  Call Extruder(12670.239)
  MoveL 1268 to (9.47, 41.51, 60) mm, rotated rx 180 ry 0 rz 180 deg; joints [36.675, 60.104, 7.721, -141.195, 72.379, -193.682]
  Call Extruder(12685.135)
  MoveL 1269 to (0, 42.57, 60) mm, rotated rx 180 ry 0 rz 180 deg; joints [37.594, 59.268, 9.663, -140.474, 73.45, -193.226]
  Call Extruder(12700.031)
  MoveL 1270 to (-9.47, 41.5, 60) mm, rotated rx -180 ry 0 rz 180 deg; joints [38.304, 58.316, 11.901, -139.989, 74.597, -192.569]
  Call Extruder(12714.927)
  MoveL 1271 to (-18.47, 38.36, 60) mm, rotated rx 180 ry 0 rz 180 deg; joints [38.762, 57.3, 14.324, -139.766, 75.77, -191.749]
  Call Extruder(12729.823)
  MoveL 1272 to (-26.54, 33.28, 60) mm, rotated rx -180 ry 0 rz 180 deg; joints [38.928, 56.273, 16.816, -139.828, 76.922, -190.815]
  Call Extruder(12744.719)
  MoveL 1273 to (-33.29, 26.54, 60) mm, rotated rx 180 ry 0 rz 180 deg; joints [38.772, 55.287, 19.256, -140.194, 78.008, -189.824]
  Call Extruder(12759.614)
  MoveL 1274 to (-38.36, 18.47, 60) mm, rotated rx 180 ry 0 rz 180 deg; joints [38.277, 54.389, 21.525, -140.869, 78.986, -188.835]
  Call Extruder(12774.510)
  MoveL 1275 to (-41.51, 9.47, 60) mm, rotated rx 180 ry 0 rz 180 deg; joints [37.447, 53.619, 23.509, -141.847, 79.813, -187.91]
  Call Extruder(12789.406)
  MoveL 1276 to (-42.57, 0, 60) mm, rotated rx 180 ry 0 rz 180 deg; joints [36.31, 53.012, 25.105, -143.096, 80.448, -187.103]
  Call Extruder(12796.960)
  MoveL 1277 to (-42.03, -4.8, 60) mm, rotated rx 180 ry 0 rz 180 deg; joints [35.612, 52.795, 25.681, -143.834, 80.653, -186.771]
  Set speed (130.0 mm/s)
  MoveL 1278 to (-54.1, -7.67, 60) mm, rotated rx 180 ry 0 rz -180 deg; joints [36.421, 51.788, 28.414, -143.176, 82.129, -185.854]
  Call Extruder(12801.033)
  Set speed (30.0 mm/s)
  MoveL 1279 to (-53.59, -12.23, 60) mm, rotated rx 180 ry 0 rz 180 deg; joints [35.732, 51.595, 28.949, -143.896, 82.336, -185.556]
  Call Extruder(12811.963)
  MoveL 1280 to (-49.53, -23.85, 60) mm, rotated rx 180 ry 0 rz 180 deg; joints [33.663, 51.321, 29.715, -146.012, 82.549, -184.997]
  Call Extruder(12822.893)
  MoveL 1281 to (-42.98, -34.27, 60) mm, rotated rx -180 ry 0 rz -180 deg; joints [31.506, 51.313, 29.737, -148.181, 82.378, -184.705]
  Call Extruder(12833.823)
  MoveL 1282 to (-34.27, -42.98, 60) mm, rotated rx -180 ry 0 rz -180 deg; joints [29.427, 51.572, 29.014, -150.24, 81.809, -184.657]
  Call Extruder(12844.754)
  MoveL 1283 to (-23.85, -49.53, 60) mm, rotated rx 180 ry 0 rz 180 deg; joints [27.581, 52.088, 27.588, -152.034, 80.86, -184.821]
  Call Extruder(12855.684)
  MoveL 1284 to (-12.23, -53.59, 60) mm, rotated rx 180 ry 0 rz 180 deg; joints [26.087, 52.846, 25.544, -153.443, 79.587, -185.162]
  Call Extruder(12866.614)
  MoveL 1285 to (0, -54.97, 60) mm, rotated rx 180 ry 0 rz 180 deg; joints [25.019, 53.817, 22.995, -154.389, 78.069, -185.66]
  Call Extruder(12870.401)
  MoveL 1286 to (4.24, -54.49, 60) mm, rotated rx 180 ry 0 rz 180 deg; joints [24.802, 54.206, 21.993, -154.553, 77.494, -185.883]
  Call Extruder(12877.544)
  MoveL 1287 to (12.23, -53.59, 60) mm, rotated rx 180 ry 0 rz 180 deg; joints [24.406, 54.961, 20.076, -154.842, 76.4, -186.302]
  Call Extruder(12888.474)
  MoveL 1288 to (23.85, -49.53, 60) mm, rotated rx -180 ry 0 rz 180 deg; joints [24.239, 56.226, 16.932, -154.807, 74.681, -187.084]
  Call Extruder(12899.405)
  MoveL 1289 to (34.27, -42.98, 60) mm, rotated rx -180 ry 0 rz 180 deg; joints [24.487, 57.553, 13.715, -154.316, 73.007, -188.001]
  Call Extruder(12910.335)
  MoveL 1290 to (42.98, -34.27, 60) mm, rotated rx 180 ry 0 rz 180 deg; joints [25.101, 58.878, 10.576, -153.422, 71.469, -189.035]
  Call Extruder(12921.265)
  MoveL 1291 to (49.52, -23.85, 60) mm, rotated rx 180 ry 0 rz 180 deg; joints [26.025, 60.129, 7.663, -152.193, 70.145, -190.155]
  Call Extruder(12932.195)
  MoveL 1292 to (53.59, -12.23, 60) mm, rotated rx -180 ry 0 rz 180 deg; joints [27.2, 61.238, 5.12, -150.706, 69.104, -191.316]
  Call Extruder(12943.125)
  MoveL 1293 to (54.97, 0, 60) mm, rotated rx 180 ry 0 rz 180 deg; joints [28.57, 62.141, 3.074, -149.045, 68.397, -192.452]
  Call Extruder(12954.056)
  MoveL 1294 to (53.59, 12.23, 60) mm, rotated rx 180 ry 0 rz 180 deg; joints [30.077, 62.781, 1.635, -147.296, 68.057, -193.492]
  Call Extruder(12964.986)
  MoveL 1295 to (49.52, 23.85, 60) mm, rotated rx 180 ry 0 rz 180 deg; joints [31.665, 63.117, 0.883, -145.541, 68.093, -194.361]
  Call Extruder(12975.916)
  MoveL 1296 to (42.98, 34.27, 60) mm, rotated rx 180 ry 0 rz 180 deg; joints [33.282, 63.127, 0.862, -143.855, 68.493, -194.991]
  Call Extruder(12986.846)
  MoveL 1297 to (34.27, 42.98, 60) mm, rotated rx 180 ry 0 rz -180 deg; joints [34.874, 62.81, 1.571, -142.299, 69.223, -195.333]
  Call Extruder(12997.776)
  MoveL 1298 to (23.85, 49.53, 60) mm, rotated rx -180 ry 0 rz 180 deg; joints [36.387, 62.186, 2.972, -140.922, 70.232, -195.357]
  Call Extruder(13008.707)
  MoveL 1299 to (12.23, 53.59, 60) mm, rotated rx 180 ry 0 rz 180 deg; joints [37.766, 61.298, 4.984, -139.762, 71.46, -195.06]
  Call Extruder(13019.637)
  MoveL 1300 to (0, 54.97, 60) mm, rotated rx 180 ry 0 rz 180 deg; joints [38.954, 60.199, 7.502, -138.852, 72.838, -194.458]
  Call Extruder(13030.567)
  MoveL 1301 to (-12.23, 53.59, 60) mm, rotated rx -180 ry 0 rz -180 deg; joints [39.895, 58.954, 10.397, -138.223, 74.302, -193.588]
  Call Extruder(13041.497)
  MoveL 1302 to (-23.85, 49.53, 60) mm, rotated rx 180 ry 0 rz 180 deg; joints [40.528, 57.632, 13.527, -137.907, 75.791, -192.502]
  Call Extruder(13052.427)
  MoveL 1303 to (-34.27, 42.98, 60) mm, rotated rx 180 ry 0 rz 180 deg; joints [40.799, 56.303, 16.743, -137.938, 77.247, -191.265]
  Call Extruder(13063.358)
  MoveL 1304 to (-42.98, 34.27, 60) mm, rotated rx 180 ry 0 rz 180 deg; joints [40.659, 55.032, 19.896, -138.348, 78.623, -189.952]
  Call Extruder(13074.288)
  MoveL 1305 to (-49.53, 23.85, 60) mm, rotated rx -180 ry 0 rz -180 deg; joints [40.072, 53.88, 22.832, -139.16, 79.87, -188.645]
  Call Extruder(13085.218)
  MoveL 1306 to (-53.59, 12.23, 60) mm, rotated rx 180 ry 0 rz 180 deg; joints [39.031, 52.898, 25.406, -140.38, 80.94, -187.427]
  Call Extruder(13096.148)
  MoveL 1307 to (-54.97, 0, 60) mm, rotated rx 180 ry 0 rz 180 deg; joints [37.56, 52.127, 27.484, -141.981, 81.781, -186.377]
  Call Extruder(13101.674)
  MoveL 1308 to (-54.27, -6.18, 60) mm, rotated rx 180 ry 0 rz -180 deg; joints [36.644, 51.852, 28.237, -142.942, 82.062, -185.954]
  Set speed (130.0 mm/s)
  MoveL 1309 to (-49.9, -9.51, 60) mm, rotated rx -180 ry 0 rz -180 deg; joints [35.741, 51.987, 27.866, -143.829, 81.779, -185.968]
  MoveL 1310 to (2.97, -12.99, 60) mm, rotated rx 180 ry 0 rz 180 deg; joints [30.614, 56.045, 17.377, -148.309, 75.785, -188.621]
  Call Extruder(13106.337)
  Set speed (80.0 mm/s)
  MoveL 1311 to (5.78, -12.01, 60) mm, rotated rx -180 ry 0 rz -180 deg; joints [30.526, 56.355, 16.616, -148.338, 75.388, -188.843]
  Call Extruder(13111.001)
  MoveL 1312 to (8.31, -10.42, 60) mm, rotated rx 180 ry 0 rz -180 deg; joints [30.538, 56.675, 15.835, -148.261, 74.998, -189.096]
  Call Extruder(13115.665)
  MoveL 1313 to (10.42, -8.31, 60) mm, rotated rx 180 ry 0 rz 180 deg; joints [30.649, 56.989, 15.074, -148.084, 74.636, -189.37]
  Call Extruder(13120.329)
  MoveL 1314 to (12.01, -5.78, 60) mm, rotated rx 180 ry 0 rz 180 deg; joints [30.85, 57.281, 14.369, -147.817, 74.319, -189.653]
  Call Extruder(13124.992)
  MoveL 1315 to (12.99, -2.97, 60) mm, rotated rx 180 ry 0 rz -180 deg; joints [31.131, 57.536, 13.756, -147.476, 74.065, -189.93]
  Call Extruder(13129.656)
  MoveL 1316 to (13.33, 0, 60) mm, rotated rx 180 ry 0 rz -180 deg; joints [31.476, 57.741, 13.266, -147.078, 73.885, -190.188]
  Call Extruder(13134.320)
  MoveL 1317 to (13, 2.97, 60) mm, rotated rx 180 ry 0 rz -180 deg; joints [31.869, 57.885, 12.924, -146.644, 73.789, -190.413]
  Call Extruder(13138.984)
  MoveL 1318 to (12.01, 5.78, 60) mm, rotated rx 180 ry 0 rz -180 deg; joints [32.292, 57.96, 12.745, -146.194, 73.78, -190.594]
  Call Extruder(13143.648)
  MoveL 1319 to (10.42, 8.31, 60) mm, rotated rx 180 ry 0 rz 180 deg; joints [32.725, 57.962, 12.74, -145.75, 73.857, -190.719]
  Call Extruder(13148.312)
  MoveL 1320 to (8.31, 10.42, 60) mm, rotated rx 180 ry 0 rz -180 deg; joints [33.149, 57.891, 12.908, -145.333, 74.017, -190.782]
  Call Extruder(13152.975)
  MoveL 1321 to (5.78, 12.01, 60) mm, rotated rx -180 ry 0 rz -180 deg; joints [33.544, 57.751, 13.242, -144.961, 74.25, -190.777]
  Call Extruder(13157.639)
  MoveL 1322 to (2.97, 13, 60) mm, rotated rx -180 ry 0 rz 180 deg; joints [33.893, 57.55, 13.724, -144.65, 74.544, -190.705]
  Call Extruder(13162.303)
  MoveL 1323 to (0, 13.33, 60) mm, rotated rx 180 ry 0 rz 180 deg; joints [34.177, 57.297, 14.33, -144.416, 74.885, -190.568]
  Call Extruder(13166.967)
  MoveL 1324 to (-2.97, 13, 60) mm, rotated rx 180 ry 0 rz 180 deg; joints [34.384, 57.007, 15.03, -144.27, 75.255, -190.375]
  Call Extruder(13171.630)
  MoveL 1325 to (-5.78, 12.01, 60) mm, rotated rx 180 ry 0 rz -180 deg; joints [34.5, 56.694, 15.79, -144.22, 75.638, -190.136]
  Call Extruder(13176.294)
  MoveL 1326 to (-8.31, 10.42, 60) mm, rotated rx 180 ry 0 rz 180 deg; joints [34.518, 56.374, 16.571, -144.269, 76.015, -189.863]
  Call Extruder(13180.958)
  MoveL 1327 to (-10.42, 8.31, 60) mm, rotated rx 180 ry 0 rz -180 deg; joints [34.436, 56.063, 17.333, -144.417, 76.368, -189.571]
  Call Extruder(13185.622)
  MoveL 1328 to (-12.01, 5.78, 60) mm, rotated rx 180 ry 0 rz 180 deg; joints [34.254, 55.776, 18.04, -144.66, 76.681, -189.278]
  Call Extruder(13190.285)
  MoveL 1329 to (-13, 2.97, 60) mm, rotated rx 180 ry 0 rz 180 deg; joints [33.981, 55.528, 18.655, -144.986, 76.938, -188.997]
  Call Extruder(13194.949)
  MoveL 1330 to (-13.33, 0, 60) mm, rotated rx -180 ry 0 rz -180 deg; joints [33.63, 55.331, 19.148, -145.382, 77.126, -188.744]
  Call Extruder(13199.613)
  MoveL 1331 to (-13, -2.97, 60) mm, rotated rx 180 ry 0 rz -180 deg; joints [33.218, 55.193, 19.493, -145.826, 77.234, -188.532]
  Call Extruder(13204.277)
  MoveL 1332 to (-12.01, -5.78, 60) mm, rotated rx 180 ry 0 rz -180 deg; joints [32.767, 55.121, 19.672, -146.297, 77.258, -188.369]
  Call Extruder(13208.941)
  MoveL 1333 to (-10.42, -8.31, 60) mm, rotated rx 180 ry 0 rz 180 deg; joints [32.302, 55.119, 19.678, -146.769, 77.193, -188.263]
  Call Extruder(13213.605)
  MoveL 1334 to (-8.31, -10.42, 60) mm, rotated rx 180 ry 0 rz -180 deg; joints [31.85, 55.187, 19.508, -147.215, 77.043, -188.218]
  Call Extruder(13218.268)
  MoveL 1335 to (-5.78, -12.01, 60) mm, rotated rx 180 ry 0 rz 180 deg; joints [31.435, 55.321, 19.172, -147.612, 76.814, -188.234]
  Call Extruder(13222.932)
  MoveL 1336 to (-2.97, -12.99, 60) mm, rotated rx 180 ry 0 rz -180 deg; joints [31.079, 55.515, 18.688, -147.937, 76.517, -188.309]
  Call Extruder(13227.596)
  MoveL 1337 to (0, -13.33, 60) mm, rotated rx -180 ry 0 rz 180 deg; joints [30.801, 55.76, 18.079, -148.173, 76.168, -188.44]
  Call Extruder(13232.260)
  MoveL 1338 to (2.97, -12.99, 60) mm, rotated rx 180 ry 0 rz 180 deg; joints [30.614, 56.045, 17.377, -148.309, 75.785, -188.621]
  Set speed (130.0 mm/s)
  MoveL 1339 to (2.97, -13, 65) mm, rotated rx -180 ry 0 rz 180 deg; joints [30.614, 55.122, 17.776, -148.238, 75.34, -188.905]
  MoveL 1340 to (-26.25, -4.54, 65) mm, rotated rx 180 ry 0 rz 180 deg; joints [34.172, 53.056, 22.883, -145.013, 78.404, -188.008]
  Call Extruder(13234.492)
  Set speed (60.0 mm/s)
  MoveL 1341 to (-26.09, -5.96, 65) mm, rotated rx 180 ry 0 rz -180 deg; joints [33.969, 52.991, 23.047, -145.23, 78.457, -187.909]
  Call Extruder(13243.857)
  MoveL 1342 to (-24.12, -11.61, 65) mm, rotated rx 180 ry 0 rz 180 deg; joints [33.033, 52.848, 23.411, -146.202, 78.513, -187.593]
  Call Extruder(13253.222)
  MoveL 1343 to (-20.93, -16.69, 65) mm, rotated rx 180 ry 0 rz -180 deg; joints [32.066, 52.844, 23.422, -147.182, 78.393, -187.393]
  Call Extruder(13262.587)
  MoveL 1344 to (-16.69, -20.93, 65) mm, rotated rx 180 ry 0 rz -180 deg; joints [31.126, 52.979, 23.078, -148.11, 78.096, -187.313]
  Call Extruder(13271.952)
  MoveL 1345 to (-11.61, -24.11, 65) mm, rotated rx 180 ry 0 rz 180 deg; joints [30.272, 53.248, 22.399, -148.931, 77.638, -187.35]
  Call Extruder(13281.317)
  MoveL 1346 to (-5.96, -26.09, 65) mm, rotated rx 180 ry 0 rz -180 deg; joints [29.552, 53.639, 21.419, -149.595, 77.039, -187.498]
  Call Extruder(13290.682)
  MoveL 1347 to (0, -26.77, 65) mm, rotated rx -180 ry 0 rz -180 deg; joints [29.003, 54.134, 20.191, -150.067, 76.332, -187.748]
  Call Extruder(13293.068)
  MoveL 1348 to (1.52, -26.59, 65) mm, rotated rx 180 ry 0 rz 180 deg; joints [28.912, 54.28, 19.832, -150.134, 76.135, -187.835]
  Call Extruder(13300.047)
  MoveL 1349 to (5.96, -26.09, 65) mm, rotated rx 180 ry 0 rz -180 deg; joints [28.65, 54.711, 18.776, -150.323, 75.556, -188.09]
  Call Extruder(13309.412)
  MoveL 1350 to (11.61, -24.12, 65) mm, rotated rx 180 ry 0 rz 180 deg; joints [28.503, 55.341, 17.247, -150.356, 74.753, -188.512]
  Call Extruder(13318.777)
  MoveL 1351 to (16.69, -20.93, 65) mm, rotated rx 180 ry 0 rz 180 deg; joints [28.559, 55.994, 15.679, -150.171, 73.968, -188.998]
  Call Extruder(13328.142)
  MoveL 1352 to (20.93, -16.69, 65) mm, rotated rx 180 ry 0 rz 180 deg; joints [28.808, 56.638, 14.15, -149.785, 73.241, -189.532]
  Call Extruder(13337.507)
  MoveL 1353 to (24.12, -11.61, 65) mm, rotated rx -180 ry 0 rz 180 deg; joints [29.229, 57.24, 12.735, -149.224, 72.612, -190.091]
  Call Extruder(13346.872)
  MoveL 1354 to (26.09, -5.96, 65) mm, rotated rx -180 ry 0 rz -180 deg; joints [29.796, 57.767, 11.505, -148.523, 72.113, -190.65]
  Call Extruder(13356.237)
  MoveL 1355 to (26.77, 0, 65) mm, rotated rx -180 ry 0 rz -180 deg; joints [30.482, 58.192, 10.52, -147.719, 71.767, -191.181]
  Call Extruder(13365.602)
  MoveL 1356 to (26.09, 5.96, 65) mm, rotated rx -180 ry 0 rz -180 deg; joints [31.252, 58.49, 9.831, -146.853, 71.591, -191.653]
  Call Extruder(13374.967)
  MoveL 1357 to (24.11, 11.61, 65) mm, rotated rx -180 ry 0 rz 180 deg; joints [32.076, 58.646, 9.472, -145.966, 71.591, -192.04]
  Call Extruder(13384.332)
  MoveL 1358 to (20.93, 16.69, 65) mm, rotated rx -180 ry 0 rz -180 deg; joints [32.917, 58.651, 9.462, -145.099, 71.763, -192.316]
  Call Extruder(13393.697)
  MoveL 1359 to (16.69, 20.93, 65) mm, rotated rx 180 ry 0 rz 180 deg; joints [33.742, 58.503, 9.8, -144.287, 72.097, -192.462]
  Call Extruder(13403.062)
  MoveL 1360 to (11.61, 24.12, 65) mm, rotated rx 180 ry 0 rz 180 deg; joints [34.517, 58.213, 10.471, -143.564, 72.571, -192.468]
  Call Extruder(13412.427)
  MoveL 1361 to (5.96, 26.09, 65) mm, rotated rx 180 ry 0 rz 180 deg; joints [35.208, 57.795, 11.439, -142.959, 73.161, -192.332]
  Call Extruder(13421.792)
  MoveL 1362 to (0, 26.77, 65) mm, rotated rx -180 ry 0 rz -180 deg; joints [35.784, 57.273, 12.657, -142.497, 73.836, -192.059]
  Call Extruder(13431.157)
  MoveL 1363 to (-5.96, 26.09, 65) mm, rotated rx 180 ry 0 rz -180 deg; joints [36.214, 56.675, 14.063, -142.2, 74.564, -191.665]
  Call Extruder(13440.522)
  MoveL 1364 to (-11.61, 24.12, 65) mm, rotated rx 180 ry 0 rz 180 deg; joints [36.473, 56.033, 15.587, -142.082, 75.312, -191.173]
  Call Extruder(13449.887)
  MoveL 1365 to (-16.69, 20.93, 65) mm, rotated rx 180 ry 0 rz -180 deg; joints [36.542, 55.379, 17.155, -142.156, 76.046, -190.611]
  Call Extruder(13459.252)
  MoveL 1366 to (-20.93, 16.69, 65) mm, rotated rx 180 ry 0 rz 180 deg; joints [36.407, 54.747, 18.689, -142.426, 76.735, -190.012]
  Call Extruder(13468.617)
  MoveL 1367 to (-24.12, 11.61, 65) mm, rotated rx -180 ry 0 rz 180 deg; joints [36.065, 54.166, 20.112, -142.889, 77.348, -189.41]
  Call Extruder(13477.982)
  MoveL 1368 to (-26.09, 5.96, 65) mm, rotated rx -180 ry 0 rz 180 deg; joints [35.528, 53.666, 21.353, -143.53, 77.856, -188.839]
  Call Extruder(13487.347)
  MoveL 1369 to (-26.77, 0, 65) mm, rotated rx 180 ry 0 rz 180 deg; joints [34.817, 53.268, 22.349, -144.323, 78.233, -188.33]
  Call Extruder(13492.135)
  MoveL 1370 to (-26.42, -3.05, 65) mm, rotated rx -180 ry 0 rz -180 deg; joints [34.385, 53.125, 22.709, -144.786, 78.348, -188.113]
  Set speed (130.0 mm/s)
  MoveL 1371 to (-41.86, -6.29, 65) mm, rotated rx 180 ry 0 rz 180 deg; joints [35.393, 51.74, 26.265, -144.007, 80.246, -187.015]
  Call Extruder(13497.133)
  Set speed (60.0 mm/s)
  MoveL 1372 to (-41.5, -9.47, 65) mm, rotated rx 180 ry 0 rz -180 deg; joints [34.924, 51.599, 26.635, -144.503, 80.375, -186.8]
  Call Extruder(13512.029)
  MoveL 1373 to (-38.36, -18.47, 65) mm, rotated rx -180 ry 0 rz 180 deg; joints [33.373, 51.376, 27.223, -146.1, 80.498, -186.33]
  Call Extruder(13526.925)
  MoveL 1374 to (-33.29, -26.54, 65) mm, rotated rx -180 ry 0 rz 180 deg; joints [31.763, 51.369, 27.24, -147.725, 80.333, -186.054]
  Call Extruder(13541.821)
  MoveL 1375 to (-26.54, -33.28, 65) mm, rotated rx 180 ry 0 rz -180 deg; joints [30.206, 51.58, 26.685, -149.265, 79.877, -185.966]
  Call Extruder(13556.716)
  MoveL 1376 to (-18.47, -38.36, 65) mm, rotated rx 180 ry 0 rz 180 deg; joints [28.808, 51.998, 25.592, -150.617, 79.146, -186.053]
  Call Extruder(13571.612)
  MoveL 1377 to (-9.47, -41.5, 65) mm, rotated rx 180 ry 0 rz -180 deg; joints [27.654, 52.609, 24.019, -151.693, 78.179, -186.296]
  Call Extruder(13586.508)
  MoveL 1378 to (0, -42.57, 65) mm, rotated rx 180 ry 0 rz 180 deg; joints [26.805, 53.386, 22.053, -152.435, 77.033, -186.681]
  Call Extruder(13591.660)
  MoveL 1379 to (3.28, -42.2, 65) mm, rotated rx -180 ry 0 rz -180 deg; joints [26.624, 53.696, 21.278, -152.569, 76.599, -186.859]
  Call Extruder(13601.404)
  MoveL 1380 to (9.47, -41.5, 65) mm, rotated rx 180 ry 0 rz 180 deg; joints [26.29, 54.294, 19.796, -152.811, 75.773, -187.195]
  Call Extruder(13616.299)
  MoveL 1381 to (18.47, -38.36, 65) mm, rotated rx 180 ry 0 rz 180 deg; joints [26.114, 55.293, 17.361, -152.817, 74.473, -187.828]
  Call Extruder(13631.195)
  MoveL 1382 to (26.54, -33.29, 65) mm, rotated rx 180 ry 0 rz 180 deg; joints [26.262, 56.335, 14.868, -152.472, 73.204, -188.565]
  Call Extruder(13646.091)
  MoveL 1383 to (33.28, -26.54, 65) mm, rotated rx 180 ry 0 rz 180 deg; joints [26.703, 57.367, 12.437, -151.81, 72.036, -189.386]
  Call Extruder(13660.987)
  MoveL 1384 to (38.36, -18.47, 65) mm, rotated rx 180 ry 0 rz -180 deg; joints [27.4, 58.336, 10.186, -150.881, 71.03, -190.264]
  Call Extruder(13675.883)
  MoveL 1385 to (41.51, -9.47, 65) mm, rotated rx 180 ry 0 rz -180 deg; joints [28.309, 59.191, 8.225, -149.742, 70.238, -191.159]
  Call Extruder(13690.779)
  MoveL 1386 to (42.57, 0, 65) mm, rotated rx 180 ry 0 rz -180 deg; joints [29.382, 59.882, 6.652, -148.457, 69.697, -192.024]
  Call Extruder(13705.674)
  MoveL 1387 to (41.5, 9.47, 65) mm, rotated rx -180 ry 0 rz 180 deg; joints [30.575, 60.37, 5.549, -147.092, 69.433, -192.808]
  Call Extruder(13720.570)
  MoveL 1388 to (38.36, 18.47, 65) mm, rotated rx -180 ry 0 rz -180 deg; joints [31.839, 60.626, 4.973, -145.711, 69.454, -193.458]
  Call Extruder(13735.466)
  MoveL 1389 to (33.28, 26.54, 65) mm, rotated rx -180 ry 0 rz -180 deg; joints [33.128, 60.633, 4.957, -144.373, 69.751, -193.93]
  Call Extruder(13750.362)
  MoveL 1390 to (26.54, 33.29, 65) mm, rotated rx 180 ry 0 rz -180 deg; joints [34.394, 60.392, 5.5, -143.13, 70.303, -194.186]
  Call Extruder(13765.258)
  MoveL 1391 to (18.47, 38.36, 65) mm, rotated rx -180 ry 0 rz 180 deg; joints [35.592, 59.917, 6.573, -142.027, 71.072, -194.208]
  Call Extruder(13780.153)
  MoveL 1392 to (9.47, 41.5, 65) mm, rotated rx 180 ry 0 rz 180 deg; joints [36.675, 59.236, 8.12, -141.101, 72.014, -193.99]
  Call Extruder(13795.049)
  MoveL 1393 to (0, 42.57, 65) mm, rotated rx -180 ry 0 rz -180 deg; joints [37.594, 58.39, 10.061, -140.382, 73.081, -193.545]
  Call Extruder(13809.945)
  MoveL 1394 to (-9.47, 41.5, 65) mm, rotated rx 180 ry 0 rz 180 deg; joints [38.304, 57.426, 12.298, -139.901, 74.221, -192.897]
  Call Extruder(13824.841)
  MoveL 1395 to (-18.47, 38.36, 65) mm, rotated rx 180 ry 0 rz 180 deg; joints [38.762, 56.396, 14.722, -139.682, 75.384, -192.086]
  Call Extruder(13839.737)
  MoveL 1396 to (-26.54, 33.29, 65) mm, rotated rx 180 ry 0 rz -180 deg; joints [38.928, 55.354, 17.215, -139.749, 76.524, -191.16]
  Call Extruder(13854.632)
  MoveL 1397 to (-33.29, 26.54, 65) mm, rotated rx 180 ry 0 rz 180 deg; joints [38.772, 54.351, 19.657, -140.119, 77.596, -190.175]
  Call Extruder(13869.528)
  MoveL 1398 to (-38.36, 18.47, 65) mm, rotated rx -180 ry 0 rz 180 deg; joints [38.277, 53.436, 21.927, -140.8, 78.559, -189.19]
  Call Extruder(13884.424)
  MoveL 1399 to (-41.51, 9.47, 65) mm, rotated rx 180 ry 0 rz -180 deg; joints [37.447, 52.65, 23.914, -141.783, 79.37, -188.265]
  Call Extruder(13899.320)
  MoveL 1400 to (-42.57, 0, 65) mm, rotated rx 180 ry 0 rz 180 deg; joints [36.31, 52.029, 25.512, -143.036, 79.988, -187.454]
  Call Extruder(13906.874)
  MoveL 1401 to (-42.03, -4.8, 65) mm, rotated rx 180 ry 0 rz 180 deg; joints [35.612, 51.807, 26.089, -143.776, 80.185, -187.118]
  Set speed (130.0 mm/s)
  MoveL 1402 to (-54.1, -7.67, 65) mm, rotated rx 180 ry 0 rz -180 deg; joints [36.421, 50.775, 28.827, -143.125, 81.649, -186.218]
  Call Extruder(13910.947)
  Set speed (30.0 mm/s)
  MoveL 1403 to (-53.59, -12.23, 65) mm, rotated rx 180 ry 0 rz -180 deg; joints [35.732, 50.577, 29.362, -143.846, 81.848, -185.915]
  Call Extruder(13921.877)
  MoveL 1404 to (-49.53, -23.85, 65) mm, rotated rx -180 ry 0 rz -180 deg; joints [33.663, 50.295, 30.131, -145.965, 82.043, -185.341]
  Call Extruder(13932.807)
  MoveL 1405 to (-42.98, -34.27, 65) mm, rotated rx 180 ry 0 rz -180 deg; joints [31.506, 50.287, 30.153, -148.136, 81.86, -185.03]
  Call Extruder(13943.737)
  MoveL 1406 to (-34.27, -42.98, 65) mm, rotated rx 180 ry 0 rz -180 deg; joints [29.427, 50.553, 29.428, -150.195, 81.284, -184.961]
  Call Extruder(13954.667)
  MoveL 1407 to (-23.85, -49.53, 65) mm, rotated rx 180 ry 0 rz 180 deg; joints [27.581, 51.084, 27.999, -151.988, 80.336, -185.103]
  Call Extruder(13965.598)
  MoveL 1408 to (-12.23, -53.59, 65) mm, rotated rx 180 ry 0 rz 180 deg; joints [26.087, 51.86, 25.951, -153.394, 79.069, -185.426]
  Call Extruder(13976.528)
  MoveL 1409 to (0, -54.97, 65) mm, rotated rx -180 ry 0 rz -180 deg; joints [25.019, 52.853, 23.399, -154.337, 77.563, -185.908]
  Call Extruder(13980.688)
  MoveL 1410 to (4.66, -54.44, 65) mm, rotated rx 180 ry 0 rz -180 deg; joints [24.781, 53.289, 22.296, -154.515, 76.937, -186.149]
  Call Extruder(13987.458)
  MoveL 1411 to (12.23, -53.59, 65) mm, rotated rx 180 ry 0 rz -180 deg; joints [24.406, 54.019, 20.477, -154.786, 75.911, -186.539]
  Call Extruder(13998.388)
  MoveL 1412 to (23.85, -49.52, 65) mm, rotated rx 180 ry 0 rz 180 deg; joints [24.239, 55.306, 17.331, -154.745, 74.21, -187.315]
  Call Extruder(14009.318)
  MoveL 1413 to (34.27, -42.98, 65) mm, rotated rx 180 ry 0 rz 180 deg; joints [24.487, 56.654, 14.113, -154.248, 72.555, -188.229]
  Call Extruder(14020.249)
  MoveL 1414 to (42.98, -34.27, 65) mm, rotated rx 180 ry 0 rz -180 deg; joints [25.101, 57.996, 10.974, -153.348, 71.036, -189.264]
  Call Extruder(14031.179)
  MoveL 1415 to (49.52, -23.85, 65) mm, rotated rx 180 ry 0 rz 180 deg; joints [26.025, 59.261, 8.063, -152.113, 69.731, -190.388]
  Call Extruder(14042.109)
  MoveL 1416 to (53.59, -12.23, 65) mm, rotated rx 180 ry 0 rz 180 deg; joints [27.2, 60.382, 5.521, -150.62, 68.708, -191.554]
  Call Extruder(14053.039)
  MoveL 1417 to (54.97, 0, 65) mm, rotated rx 180 ry 0 rz 180 deg; joints [28.57, 61.293, 3.478, -148.954, 68.016, -192.699]
  Call Extruder(14063.969)
  MoveL 1418 to (53.59, 12.23, 65) mm, rotated rx 180 ry 0 rz -180 deg; joints [30.077, 61.939, 2.041, -147.2, 67.689, -193.748]
  Call Extruder(14074.900)
  MoveL 1419 to (49.52, 23.85, 65) mm, rotated rx 180 ry 0 rz 180 deg; joints [31.665, 62.277, 1.29, -145.442, 67.736, -194.626]
  Call Extruder(14085.830)
  MoveL 1420 to (42.98, 34.27, 65) mm, rotated rx 180 ry 0 rz 180 deg; joints [33.282, 62.287, 1.268, -143.753, 68.143, -195.266]
  Call Extruder(14096.760)
  MoveL 1421 to (34.27, 42.98, 65) mm, rotated rx 180 ry 0 rz -180 deg; joints [34.874, 61.967, 1.977, -142.196, 68.878, -195.619]
  Call Extruder(14107.690)
  MoveL 1422 to (23.85, 49.53, 65) mm, rotated rx 180 ry 0 rz -180 deg; joints [36.387, 61.339, 3.375, -140.82, 69.888, -195.655]
  Call Extruder(14118.620)
  MoveL 1423 to (12.23, 53.59, 65) mm, rotated rx 180 ry 0 rz -180 deg; joints [37.766, 60.442, 5.386, -139.663, 71.113, -195.37]
  Call Extruder(14129.551)
  MoveL 1424 to (0, 54.97, 65) mm, rotated rx 180 ry 0 rz 180 deg; joints [38.954, 59.332, 7.902, -138.756, 72.487, -194.781]
  Call Extruder(14140.481)
  MoveL 1425 to (-12.23, 53.59, 65) mm, rotated rx -180 ry 0 rz 180 deg; joints [39.895, 58.073, 10.795, -138.132, 73.942, -193.923]
  Call Extruder(14151.411)
  MoveL 1426 to (-23.85, 49.53, 65) mm, rotated rx 180 ry 0 rz 180 deg; joints [40.528, 56.734, 13.924, -137.821, 75.419, -192.849]
  Call Extruder(14162.341)
  MoveL 1427 to (-34.27, 42.98, 65) mm, rotated rx 180 ry 0 rz -180 deg; joints [40.799, 55.384, 17.142, -137.858, 76.862, -191.623]
  Call Extruder(14173.271)
  MoveL 1428 to (-42.98, 34.27, 65) mm, rotated rx 180 ry 0 rz 180 deg; joints [40.659, 54.092, 20.296, -138.274, 78.22, -190.319]
  Call Extruder(14184.202)
  MoveL 1429 to (-49.53, 23.85, 65) mm, rotated rx -180 ry 0 rz -180 deg; joints [40.072, 52.917, 23.236, -139.093, 79.447, -189.017]
  Call Extruder(14195.132)
  MoveL 1430 to (-53.59, 12.23, 65) mm, rotated rx 180 ry 0 rz 180 deg; joints [39.031, 51.913, 25.814, -140.32, 80.495, -187.801]
  Call Extruder(14206.062)
  MoveL 1431 to (-54.97, 0, 65) mm, rotated rx 180 ry 0 rz -180 deg; joints [37.56, 51.123, 27.895, -141.927, 81.314, -186.747]
  Call Extruder(14211.588)
  MoveL 1432 to (-54.27, -6.18, 65) mm, rotated rx 180 ry 0 rz -180 deg; joints [36.644, 50.841, 28.649, -142.89, 81.584, -186.318]
  Set speed (130.0 mm/s)
  MoveL 1433 to (-49.9, -9.51, 65) mm, rotated rx -180 ry 0 rz -180 deg; joints [35.741, 50.979, 28.278, -143.777, 81.298, -186.324]
  MoveL 1434 to (0.02, -13.33, 65) mm, rotated rx 180 ry 0 rz 180 deg; joints [30.8, 54.835, 18.473, -148.104, 75.717, -188.729]
  Call Extruder(14216.216)
  Set speed (80.0 mm/s)
  MoveL 1435 to (2.97, -13, 65) mm, rotated rx -180 ry 0 rz 180 deg; joints [30.614, 55.122, 17.776, -148.238, 75.34, -188.905]
  Call Extruder(14220.880)
  MoveL 1436 to (5.78, -12.01, 65) mm, rotated rx 180 ry 0 rz -180 deg; joints [30.526, 55.437, 17.015, -148.266, 74.947, -189.125]
  Call Extruder(14225.543)
  MoveL 1437 to (8.31, -10.42, 65) mm, rotated rx 180 ry 0 rz -180 deg; joints [30.538, 55.762, 16.234, -148.188, 74.561, -189.377]
  Call Extruder(14230.208)
  MoveL 1438 to (10.42, -8.31, 65) mm, rotated rx 180 ry 0 rz -180 deg; joints [30.649, 56.081, 15.472, -148.009, 74.203, -189.651]
  Call Extruder(14234.871)
  MoveL 1439 to (12.01, -5.78, 65) mm, rotated rx 180 ry 0 rz 180 deg; joints [30.85, 56.378, 14.767, -147.741, 73.891, -189.933]
  Call Extruder(14239.535)
  MoveL 1440 to (12.99, -2.97, 65) mm, rotated rx -180 ry 0 rz 180 deg; joints [31.131, 56.636, 14.154, -147.398, 73.642, -190.211]
  Call Extruder(14244.199)
  MoveL 1441 to (13.33, 0, 65) mm, rotated rx 180 ry 0 rz -180 deg; joints [31.476, 56.844, 13.664, -146.999, 73.466, -190.471]
  Call Extruder(14248.863)
  MoveL 1442 to (13, 2.97, 65) mm, rotated rx -180 ry 0 rz -180 deg; joints [31.869, 56.99, 13.321, -146.563, 73.374, -190.699]
  Call Extruder(14253.526)
  MoveL 1443 to (12.01, 5.78, 65) mm, rotated rx 180 ry 0 rz 180 deg; joints [32.292, 57.066, 13.143, -146.113, 73.368, -190.882]
  Call Extruder(14258.190)
  MoveL 1444 to (10.42, 8.31, 65) mm, rotated rx 180 ry 0 rz 180 deg; joints [32.725, 57.068, 13.137, -145.668, 73.447, -191.011]
  Call Extruder(14262.854)
  MoveL 1445 to (8.31, 10.42, 65) mm, rotated rx 180 ry 0 rz 180 deg; joints [33.149, 56.996, 13.306, -145.251, 73.608, -191.076]
  Call Extruder(14267.518)
  MoveL 1446 to (5.78, 12.01, 65) mm, rotated rx 180 ry 0 rz -180 deg; joints [33.544, 56.854, 13.64, -144.879, 73.841, -191.075]
  Call Extruder(14272.181)
  MoveL 1447 to (2.97, 13, 65) mm, rotated rx 180 ry 0 rz -180 deg; joints [33.893, 56.65, 14.121, -144.569, 74.135, -191.007]
  Call Extruder(14276.845)
  MoveL 1448 to (0, 13.33, 65) mm, rotated rx 180 ry 0 rz 180 deg; joints [34.177, 56.394, 14.728, -144.336, 74.474, -190.874]
  Call Extruder(14281.509)
  MoveL 1449 to (-2.97, 13, 65) mm, rotated rx 180 ry 0 rz 180 deg; joints [34.384, 56.099, 15.428, -144.191, 74.842, -190.684]
  Call Extruder(14286.173)
  MoveL 1450 to (-5.78, 12.01, 65) mm, rotated rx 180 ry 0 rz -180 deg; joints [34.5, 55.781, 16.188, -144.142, 75.221, -190.446]
  Call Extruder(14290.836)
  MoveL 1451 to (-8.31, 10.42, 65) mm, rotated rx 180 ry 0 rz -180 deg; joints [34.518, 55.456, 16.969, -144.192, 75.594, -190.175]
  Call Extruder(14295.501)
  MoveL 1452 to (-10.42, 8.31, 65) mm, rotated rx 180 ry 0 rz 180 deg; joints [34.436, 55.14, 17.732, -144.342, 75.942, -189.886]
  Call Extruder(14300.164)
  MoveL 1453 to (-12.01, 5.78, 65) mm, rotated rx 180 ry 0 rz -180 deg; joints [34.254, 54.849, 18.439, -144.586, 76.25, -189.592]
  Call Extruder(14304.828)
  MoveL 1454 to (-13, 2.97, 65) mm, rotated rx 180 ry 0 rz 180 deg; joints [33.981, 54.597, 19.055, -144.914, 76.502, -189.311]
  Call Extruder(14309.492)
  MoveL 1455 to (-13.33, 0, 65) mm, rotated rx -180 ry 0 rz -180 deg; joints [33.63, 54.395, 19.548, -145.311, 76.685, -189.057]
  Call Extruder(14314.156)
  MoveL 1456 to (-13, -2.97, 65) mm, rotated rx -180 ry 0 rz -180 deg; joints [33.218, 54.255, 19.893, -145.757, 76.79, -188.842]
  Call Extruder(14318.819)
  MoveL 1457 to (-12.01, -5.78, 65) mm, rotated rx 180 ry 0 rz -180 deg; joints [32.767, 54.182, 20.073, -146.228, 76.81, -188.676]
  Call Extruder(14323.483)
  MoveL 1458 to (-10.42, -8.31, 65) mm, rotated rx 180 ry 0 rz 180 deg; joints [32.302, 54.18, 20.078, -146.7, 76.743, -188.566]
  Call Extruder(14328.147)
  MoveL 1459 to (-8.31, -10.42, 65) mm, rotated rx 180 ry 0 rz -180 deg; joints [31.85, 54.249, 19.908, -147.147, 76.591, -188.517]
  Call Extruder(14332.811)
  MoveL 1460 to (-5.78, -12.01, 65) mm, rotated rx -180 ry 0 rz -180 deg; joints [31.435, 54.385, 19.572, -147.543, 76.362, -188.529]
  Call Extruder(14337.474)
  MoveL 1461 to (-2.97, -12.99, 65) mm, rotated rx 180 ry 0 rz 180 deg; joints [31.079, 54.583, 19.088, -147.868, 76.066, -188.6]
  Call Extruder(14342.173)
  MoveL 1462 to (0.02, -13.33, 65) mm, rotated rx 180 ry 0 rz 180 deg; joints [30.8, 54.835, 18.473, -148.104, 75.717, -188.729]
  Set speed (130.0 mm/s)
  MoveL 1463 to (0.02, -13.33, 70) mm, rotated rx -180 ry 0 rz -180 deg; joints [30.8, 53.912, 18.855, -148.03, 75.258, -189.025]
  MoveL 1464 to (-26.25, -4.54, 70) mm, rotated rx 180 ry 0 rz 180 deg; joints [34.172, 52.1, 23.269, -144.945, 77.937, -188.342]
  Call Extruder(14344.405)
  Set speed (60.0 mm/s)
  MoveL 1465 to (-26.09, -5.96, 70) mm, rotated rx 180 ry 0 rz 180 deg; joints [33.969, 52.033, 23.434, -145.162, 77.988, -188.242]
  Call Extruder(14353.770)
  MoveL 1466 to (-24.12, -11.61, 70) mm, rotated rx 180 ry 0 rz 180 deg; joints [33.033, 51.887, 23.798, -146.136, 78.037, -187.919]
  Call Extruder(14363.135)
  MoveL 1467 to (-20.93, -16.69, 70) mm, rotated rx -180 ry 0 rz 180 deg; joints [32.066, 51.883, 23.809, -147.117, 77.91, -187.711]
  Call Extruder(14372.500)
  MoveL 1468 to (-16.69, -20.93, 70) mm, rotated rx -180 ry 0 rz -180 deg; joints [31.126, 52.021, 23.465, -148.045, 77.611, -187.622]
  Call Extruder(14381.865)
  MoveL 1469 to (-11.61, -24.11, 70) mm, rotated rx 180 ry 0 rz 180 deg; joints [30.272, 52.296, 22.784, -148.866, 77.152, -187.65]
  Call Extruder(14391.230)
  MoveL 1470 to (-5.96, -26.09, 70) mm, rotated rx -180 ry 0 rz -180 deg; joints [29.552, 52.694, 21.804, -149.529, 76.556, -187.79]
  Call Extruder(14400.595)
  MoveL 1471 to (0, -26.77, 70) mm, rotated rx 180 ry 0 rz 180 deg; joints [29.003, 53.199, 20.574, -149.999, 75.854, -188.032]
  Call Extruder(14403.637)
  MoveL 1472 to (1.94, -26.55, 70) mm, rotated rx 180 ry 0 rz 180 deg; joints [28.887, 53.388, 20.117, -150.083, 75.605, -188.141]
  Call Extruder(14409.960)
  MoveL 1473 to (5.96, -26.09, 70) mm, rotated rx -180 ry 0 rz 180 deg; joints [28.65, 53.785, 19.158, -150.253, 75.084, -188.368]
  Call Extruder(14419.325)
  MoveL 1474 to (11.61, -24.12, 70) mm, rotated rx 180 ry 0 rz 180 deg; joints [28.503, 54.426, 17.628, -150.283, 74.29, -188.786]
  Call Extruder(14428.690)
  MoveL 1475 to (16.69, -20.93, 70) mm, rotated rx -180 ry 0 rz -180 deg; joints [28.559, 55.09, 16.06, -150.095, 73.514, -189.27]
  Call Extruder(14438.055)
  MoveL 1476 to (20.93, -16.69, 70) mm, rotated rx -180 ry 0 rz -180 deg; joints [28.808, 55.743, 14.53, -149.706, 72.797, -189.803]
  Call Extruder(14447.420)
  MoveL 1477 to (24.12, -11.61, 70) mm, rotated rx 180 ry 0 rz 180 deg; joints [29.229, 56.353, 13.115, -149.142, 72.178, -190.363]
  Call Extruder(14456.785)
  MoveL 1478 to (26.09, -5.96, 70) mm, rotated rx 180 ry 0 rz -180 deg; joints [29.796, 56.887, 11.885, -148.438, 71.687, -190.925]
  Call Extruder(14466.150)
  MoveL 1479 to (26.77, 0, 70) mm, rotated rx 180 ry 0 rz 180 deg; joints [30.482, 57.317, 10.901, -147.631, 71.35, -191.459]
  Call Extruder(14475.515)
  MoveL 1480 to (26.09, 5.96, 70) mm, rotated rx -180 ry 0 rz -180 deg; joints [31.252, 57.619, 10.212, -146.762, 71.181, -191.936]
  Call Extruder(14484.880)
  MoveL 1481 to (24.11, 11.61, 70) mm, rotated rx 180 ry 0 rz -180 deg; joints [32.076, 57.777, 9.853, -145.874, 71.187, -192.328]
  Call Extruder(14494.245)
  MoveL 1482 to (20.93, 16.69, 70) mm, rotated rx -180 ry 0 rz -180 deg; joints [32.917, 57.782, 9.843, -145.006, 71.364, -192.61]
  Call Extruder(14503.610)
  MoveL 1483 to (16.69, 20.93, 70) mm, rotated rx -180 ry 0 rz 180 deg; joints [33.742, 57.633, 10.181, -144.193, 71.7, -192.763]
  Call Extruder(14512.975)
  MoveL 1484 to (11.61, 24.12, 70) mm, rotated rx 180 ry 0 rz -180 deg; joints [34.517, 57.339, 10.852, -143.471, 72.175, -192.776]
  Call Extruder(14522.340)
  MoveL 1485 to (5.96, 26.09, 70) mm, rotated rx 180 ry 0 rz -180 deg; joints [35.208, 56.916, 11.82, -142.867, 72.763, -192.646]
  Call Extruder(14531.705)
  MoveL 1486 to (0, 26.77, 70) mm, rotated rx 180 ry 0 rz 180 deg; joints [35.784, 56.387, 13.037, -142.407, 73.435, -192.38]
  Call Extruder(14541.070)
  MoveL 1487 to (-5.96, 26.09, 70) mm, rotated rx 180 ry 0 rz 180 deg; joints [36.214, 55.781, 14.443, -142.111, 74.158, -191.993]
  Call Extruder(14550.435)
  MoveL 1488 to (-11.61, 24.12, 70) mm, rotated rx 180 ry 0 rz -180 deg; joints [36.473, 55.129, 15.968, -141.996, 74.899, -191.506]
  Call Extruder(14559.800)
  MoveL 1489 to (-16.69, 20.93, 70) mm, rotated rx -180 ry 0 rz 180 deg; joints [36.542, 54.465, 17.536, -142.074, 75.626, -190.948]
  Call Extruder(14569.165)
  MoveL 1490 to (-20.93, 16.69, 70) mm, rotated rx -180 ry 0 rz 180 deg; joints [36.407, 53.822, 19.071, -142.347, 76.305, -190.352]
  Call Extruder(14578.530)
  MoveL 1491 to (-24.12, 11.61, 70) mm, rotated rx 180 ry 0 rz -180 deg; joints [36.065, 53.231, 20.496, -142.813, 76.908, -189.751]
  Call Extruder(14587.894)
  MoveL 1492 to (-26.09, 5.96, 70) mm, rotated rx 180 ry 0 rz -180 deg; joints [35.528, 52.721, 21.738, -143.457, 77.406, -189.18]
  Call Extruder(14597.260)
  MoveL 1493 to (-26.77, 0, 70) mm, rotated rx 180 ry 0 rz 180 deg; joints [34.817, 52.316, 22.735, -144.253, 77.773, -188.668]
  Call Extruder(14602.048)
  MoveL 1494 to (-26.42, -3.05, 70) mm, rotated rx 180 ry 0 rz -180 deg; joints [34.385, 52.17, 23.095, -144.717, 77.883, -188.448]
  Set speed (130.0 mm/s)
  MoveL 1495 to (-41.86, -6.29, 70) mm, rotated rx -180 ry 0 rz 180 deg; joints [35.393, 50.754, 26.656, -143.946, 79.765, -187.37]
  Call Extruder(14607.046)
  Set speed (60.0 mm/s)
  MoveL 1496 to (-41.5, -9.47, 70) mm, rotated rx -180 ry 0 rz -180 deg; joints [34.924, 50.61, 27.027, -144.443, 79.889, -187.152]
  Call Extruder(14621.942)
  MoveL 1497 to (-38.36, -18.47, 70) mm, rotated rx 180 ry 0 rz -180 deg; joints [33.373, 50.381, 27.615, -146.042, 79.998, -186.671]
  Call Extruder(14636.838)
  MoveL 1498 to (-33.29, -26.54, 70) mm, rotated rx 180 ry 0 rz -180 deg; joints [31.763, 50.375, 27.632, -147.668, 79.824, -186.38]
  Call Extruder(14651.733)
  MoveL 1499 to (-26.54, -33.28, 70) mm, rotated rx -180 ry 0 rz -180 deg; joints [30.206, 50.59, 27.077, -149.209, 79.363, -186.277]
  Call Extruder(14666.629)
  MoveL 1500 to (-18.47, -38.36, 70) mm, rotated rx -180 ry 0 rz -180 deg; joints [28.808, 51.019, 25.982, -150.56, 78.632, -186.348]
  Call Extruder(14681.525)
  MoveL 1501 to (-9.47, -41.5, 70) mm, rotated rx 180 ry 0 rz 180 deg; joints [27.654, 51.643, 24.407, -151.635, 77.67, -186.577]
  Call Extruder(14696.421)
  MoveL 1502 to (0, -42.57, 70) mm, rotated rx 180 ry 0 rz 180 deg; joints [26.805, 52.436, 22.439, -152.374, 76.532, -186.95]
  Call Extruder(14702.229)
  MoveL 1503 to (3.69, -42.16, 70) mm, rotated rx 180 ry 0 rz 180 deg; joints [26.601, 52.792, 21.564, -152.523, 76.048, -187.147]
  Call Extruder(14711.317)
  MoveL 1504 to (9.47, -41.5, 70) mm, rotated rx 180 ry 0 rz 180 deg; joints [26.29, 53.362, 20.179, -152.746, 75.284, -187.455]
  Call Extruder(14726.212)
  MoveL 1505 to (18.47, -38.36, 70) mm, rotated rx 180 ry 0 rz 180 deg; joints [26.114, 54.378, 17.743, -152.748, 73.998, -188.081]
  Call Extruder(14741.108)
  MoveL 1506 to (26.54, -33.29, 70) mm, rotated rx 180 ry 0 rz 180 deg; joints [26.262, 55.436, 15.249, -152.398, 72.745, -188.816]
  Call Extruder(14756.004)
  MoveL 1507 to (33.28, -26.54, 70) mm, rotated rx -180 ry 0 rz 180 deg; joints [26.703, 56.482, 12.817, -151.732, 71.592, -189.637]
  Call Extruder(14770.900)
  MoveL 1508 to (38.36, -18.47, 70) mm, rotated rx -180 ry 0 rz -180 deg; joints [27.4, 57.464, 10.566, -150.797, 70.601, -190.517]
  Call Extruder(14785.796)
  MoveL 1509 to (41.5, -9.47, 70) mm, rotated rx -180 ry 0 rz 180 deg; joints [28.309, 58.328, 8.606, -149.654, 69.822, -191.417]
  Call Extruder(14800.691)
  MoveL 1510 to (42.57, 0, 70) mm, rotated rx 180 ry 0 rz -180 deg; joints [29.382, 59.027, 7.035, -148.364, 69.295, -192.288]
  Call Extruder(14815.587)
  MoveL 1511 to (41.5, 9.47, 70) mm, rotated rx -180 ry 0 rz -180 deg; joints [30.575, 59.52, 5.933, -146.996, 69.042, -193.079]
  Call Extruder(14830.483)
  MoveL 1512 to (38.36, 18.47, 70) mm, rotated rx 180 ry 0 rz -180 deg; joints [31.839, 59.778, 5.358, -145.612, 69.071, -193.738]
  Call Extruder(14845.379)
  MoveL 1513 to (33.28, 26.54, 70) mm, rotated rx -180 ry 0 rz 180 deg; joints [33.128, 59.785, 5.341, -144.272, 69.375, -194.218]
  Call Extruder(14860.275)
  MoveL 1514 to (26.54, 33.28, 70) mm, rotated rx -180 ry 0 rz 180 deg; joints [34.394, 59.542, 5.883, -143.029, 69.93, -194.484]
  Call Extruder(14875.170)
  MoveL 1515 to (18.47, 38.36, 70) mm, rotated rx 180 ry 0 rz 180 deg; joints [35.592, 59.062, 6.956, -141.926, 70.7, -194.516]
  Call Extruder(14890.066)
  MoveL 1516 to (9.47, 41.51, 70) mm, rotated rx 180 ry 0 rz 180 deg; joints [36.675, 58.374, 8.502, -141.001, 71.641, -194.308]
  Call Extruder(14904.962)
  MoveL 1517 to (0, 42.57, 70) mm, rotated rx 180 ry 0 rz 180 deg; joints [37.594, 57.518, 10.442, -140.286, 72.703, -193.873]
  Call Extruder(14919.858)
  MoveL 1518 to (-9.47, 41.5, 70) mm, rotated rx 180 ry 0 rz 180 deg; joints [38.304, 56.542, 12.679, -139.808, 73.836, -193.235]
  Call Extruder(14934.754)
  MoveL 1519 to (-18.47, 38.36, 70) mm, rotated rx 180 ry 0 rz -180 deg; joints [38.762, 55.498, 15.103, -139.593, 74.99, -192.433]
  Call Extruder(14949.649)
  MoveL 1520 to (-26.54, 33.29, 70) mm, rotated rx 180 ry 0 rz -180 deg; joints [38.928, 54.44, 17.596, -139.665, 76.118, -191.515]
  Call Extruder(14964.545)
  MoveL 1521 to (-33.29, 26.54, 70) mm, rotated rx -180 ry 0 rz 180 deg; joints [38.772, 53.419, 20.04, -140.041, 77.176, -190.536]
  Call Extruder(14979.441)
  MoveL 1522 to (-38.36, 18.47, 70) mm, rotated rx 180 ry 0 rz 180 deg; joints [38.277, 52.487, 22.313, -140.727, 78.122, -189.554]
  Call Extruder(14994.337)
  MoveL 1523 to (-41.51, 9.47, 70) mm, rotated rx -180 ry 0 rz -180 deg; joints [37.447, 51.685, 24.301, -141.714, 78.916, -188.629]
  Call Extruder(15009.233)
  MoveL 1524 to (-42.57, 0, 70) mm, rotated rx 180 ry 0 rz -180 deg; joints [36.31, 51.05, 25.902, -142.972, 79.518, -187.814]
  Call Extruder(15016.787)
  MoveL 1525 to (-42.03, -4.8, 70) mm, rotated rx 180 ry 0 rz -180 deg; joints [35.612, 50.823, 26.48, -143.714, 79.707, -187.474]
  Set speed (130.0 mm/s)
  MoveL 1526 to (-54.1, -7.67, 70) mm, rotated rx 180 ry 0 rz -180 deg; joints [36.421, 49.765, 29.223, -143.069, 81.158, -186.591]
  Call Extruder(15020.860)
  Set speed (30.0 mm/s)
  MoveL 1527 to (-53.59, -12.23, 70) mm, rotated rx 180 ry 0 rz -180 deg; joints [35.732, 49.561, 29.759, -143.792, 81.348, -186.285]
  Call Extruder(15031.790)
  MoveL 1528 to (-49.53, -23.85, 70) mm, rotated rx 180 ry 0 rz -180 deg; joints [33.663, 49.272, 30.529, -145.915, 81.525, -185.695]
  Call Extruder(15042.720)
  MoveL 1529 to (-42.98, -34.27, 70) mm, rotated rx 180 ry 0 rz 180 deg; joints [31.506, 49.264, 30.551, -148.088, 81.329, -185.364]
  Call Extruder(15053.650)
  MoveL 1530 to (-34.27, -42.98, 70) mm, rotated rx 180 ry 0 rz 180 deg; joints [29.427, 49.537, 29.825, -150.146, 80.747, -185.273]
  Call Extruder(15064.580)
  MoveL 1531 to (-23.85, -49.52, 70) mm, rotated rx -180 ry 0 rz -180 deg; joints [27.581, 50.082, 28.393, -151.938, 79.799, -185.393]
  Call Extruder(15075.510)
  MoveL 1532 to (-12.23, -53.59, 70) mm, rotated rx 180 ry 0 rz -180 deg; joints [26.087, 50.877, 26.342, -153.341, 78.54, -185.696]
  Call Extruder(15086.441)
  MoveL 1533 to (0, -54.97, 70) mm, rotated rx 180 ry 0 rz 180 deg; joints [25.019, 51.892, 23.786, -154.281, 77.046, -186.163]
  Call Extruder(15090.974)
  MoveL 1534 to (5.07, -54.4, 70) mm, rotated rx 180 ry 0 rz 180 deg; joints [24.76, 52.377, 22.582, -154.472, 76.371, -186.421]
  Call Extruder(15097.371)
  MoveL 1535 to (12.23, -53.59, 70) mm, rotated rx -180 ry 0 rz 180 deg; joints [24.406, 53.081, 20.86, -154.725, 75.41, -186.783]
  Call Extruder(15108.301)
  MoveL 1536 to (23.85, -49.52, 70) mm, rotated rx 180 ry 0 rz -180 deg; joints [24.239, 54.391, 17.713, -154.679, 73.727, -187.552]
  Call Extruder(15119.231)
  MoveL 1537 to (34.27, -42.98, 70) mm, rotated rx 180 ry 0 rz 180 deg; joints [24.487, 55.759, 14.493, -154.177, 72.092, -188.463]
  Call Extruder(15130.161)
  MoveL 1538 to (42.98, -34.27, 70) mm, rotated rx 180 ry 0 rz 180 deg; joints [25.101, 57.119, 11.354, -153.271, 70.593, -189.499]
  Call Extruder(15141.092)
  MoveL 1539 to (49.52, -23.85, 70) mm, rotated rx 180 ry 0 rz -180 deg; joints [26.025, 58.4, 8.444, -152.029, 69.307, -190.628]
  Call Extruder(15152.022)
  MoveL 1540 to (53.59, -12.23, 70) mm, rotated rx -180 ry 0 rz 180 deg; joints [27.2, 59.532, 5.905, -150.53, 68.301, -191.801]
  Call Extruder(15162.952)
  MoveL 1541 to (54.97, 0, 70) mm, rotated rx 180 ry 0 rz 180 deg; joints [28.57, 60.452, 3.863, -148.858, 67.626, -192.953]
  Call Extruder(15173.882)
  MoveL 1542 to (53.59, 12.23, 70) mm, rotated rx 180 ry 0 rz 180 deg; joints [30.077, 61.103, 2.428, -147.099, 67.312, -194.011]
  Call Extruder(15184.812)
  MoveL 1543 to (49.52, 23.85, 70) mm, rotated rx 180 ry 0 rz -180 deg; joints [31.665, 61.444, 1.678, -145.337, 67.37, -194.899]
  Call Extruder(15195.743)
  MoveL 1544 to (42.98, 34.27, 70) mm, rotated rx -180 ry 0 rz 180 deg; joints [33.282, 61.454, 1.657, -143.647, 67.785, -195.551]
  Call Extruder(15206.673)
  MoveL 1545 to (34.27, 42.98, 70) mm, rotated rx 180 ry 0 rz 180 deg; joints [34.874, 61.132, 2.364, -142.089, 68.524, -195.914]
  Call Extruder(15217.603)
  MoveL 1546 to (23.85, 49.53, 70) mm, rotated rx 180 ry 0 rz -180 deg; joints [36.387, 60.498, 3.761, -140.714, 69.535, -195.962]
  Call Extruder(15228.533)
  MoveL 1547 to (12.23, 53.59, 70) mm, rotated rx 180 ry 0 rz -180 deg; joints [37.766, 59.593, 5.769, -139.558, 70.758, -195.689]
  Call Extruder(15239.463)
  MoveL 1548 to (0, 54.97, 70) mm, rotated rx 180 ry 0 rz 180 deg; joints [38.954, 58.471, 8.283, -138.656, 72.127, -195.112]
  Call Extruder(15250.394)
  MoveL 1549 to (-12.23, 53.59, 70) mm, rotated rx 180 ry 0 rz 180 deg; joints [39.895, 57.197, 11.175, -138.035, 73.574, -194.268]
  Call Extruder(15261.324)
  MoveL 1550 to (-23.85, 49.52, 70) mm, rotated rx -180 ry 0 rz 180 deg; joints [40.528, 55.84, 14.305, -137.73, 75.039, -193.206]
  Call Extruder(15272.254)
  MoveL 1551 to (-34.27, 42.98, 70) mm, rotated rx 180 ry 0 rz 180 deg; joints [40.799, 54.47, 17.524, -137.773, 76.467, -191.991]
  Call Extruder(15283.184)
  MoveL 1552 to (-42.98, 34.27, 70) mm, rotated rx 180 ry 0 rz 180 deg; joints [40.659, 53.155, 20.68, -138.196, 77.807, -190.695]
  Call Extruder(15294.115)
  MoveL 1553 to (-49.53, 23.85, 70) mm, rotated rx -180 ry 0 rz 180 deg; joints [40.072, 51.957, 23.623, -139.022, 79.014, -189.399]
  Call Extruder(15305.045)
  MoveL 1554 to (-53.59, 12.23, 70) mm, rotated rx 180 ry 0 rz 180 deg; joints [39.031, 50.931, 26.204, -140.255, 80.04, -188.184]
  Call Extruder(15315.975)
  MoveL 1555 to (-54.97, 0, 70) mm, rotated rx -180 ry 0 rz 180 deg; joints [37.56, 50.122, 28.289, -141.868, 80.836, -187.126]
  Call Extruder(15321.501)
  MoveL 1556 to (-54.27, -6.18, 70) mm, rotated rx 180 ry 0 rz 180 deg; joints [36.644, 49.833, 29.044, -142.834, 81.096, -186.693]
  Set speed (130.0 mm/s)
  MoveL 1557 to (-49.9, -9.51, 70) mm, rotated rx 180 ry 0 rz 180 deg; joints [35.741, 49.975, 28.672, -143.72, 80.806, -186.689]
  MoveL 1558 to (0.44, -13.28, 70) mm, rotated rx 180 ry 0 rz 180 deg; joints [30.773, 53.953, 18.757, -148.049, 75.205, -189.049]
  Call Extruder(15325.473)
  Set speed (80.0 mm/s)
  MoveL 1559 to (2.97, -12.99, 70) mm, rotated rx 180 ry 0 rz 180 deg; joints [30.614, 54.204, 18.157, -148.163, 74.884, -189.198]
  Call Extruder(15330.137)
  MoveL 1560 to (5.78, -12.01, 70) mm, rotated rx 180 ry 0 rz 180 deg; joints [30.526, 54.524, 17.396, -148.189, 74.495, -189.415]
  Call Extruder(15334.800)
  MoveL 1561 to (8.31, -10.42, 70) mm, rotated rx 180 ry 0 rz 180 deg; joints [30.538, 54.854, 16.615, -148.11, 74.113, -189.666]
  Call Extruder(15339.464)
  MoveL 1562 to (10.42, -8.31, 70) mm, rotated rx 180 ry 0 rz 180 deg; joints [30.649, 55.178, 15.853, -147.929, 73.76, -189.939]
  Call Extruder(15344.128)
  MoveL 1563 to (12.01, -5.78, 70) mm, rotated rx 180 ry 0 rz -180 deg; joints [30.85, 55.479, 15.147, -147.659, 73.454, -190.222]
  Call Extruder(15348.792)
  MoveL 1564 to (12.99, -2.97, 70) mm, rotated rx 180 ry 0 rz -180 deg; joints [31.131, 55.741, 14.535, -147.315, 73.209, -190.501]
  Call Extruder(15353.456)
  MoveL 1565 to (13.33, 0, 70) mm, rotated rx 180 ry 0 rz -180 deg; joints [31.476, 55.952, 14.044, -146.915, 73.038, -190.762]
  Call Extruder(15358.120)
  MoveL 1566 to (13, 2.97, 70) mm, rotated rx 180 ry 0 rz -180 deg; joints [31.869, 56.1, 13.702, -146.478, 72.949, -190.992]
  Call Extruder(15362.783)
  MoveL 1567 to (12.01, 5.78, 70) mm, rotated rx 180 ry 0 rz 180 deg; joints [32.292, 56.177, 13.523, -146.027, 72.946, -191.179]
  Call Extruder(15367.447)
  MoveL 1568 to (10.42, 8.31, 70) mm, rotated rx 180 ry 0 rz 180 deg; joints [32.725, 56.179, 13.518, -145.582, 73.028, -191.31]
  Call Extruder(15372.111)
  MoveL 1569 to (8.31, 10.42, 70) mm, rotated rx 180 ry 0 rz 180 deg; joints [33.149, 56.106, 13.686, -145.164, 73.19, -191.38]
  Call Extruder(15376.775)
  MoveL 1570 to (5.78, 12.01, 70) mm, rotated rx 180 ry 0 rz -180 deg; joints [33.544, 55.963, 14.02, -144.792, 73.423, -191.382]
  Call Extruder(15381.438)
  MoveL 1571 to (2.97, 13, 70) mm, rotated rx 180 ry 0 rz -180 deg; joints [33.893, 55.755, 14.502, -144.483, 73.716, -191.317]
  Call Extruder(15386.102)
  MoveL 1572 to (0, 13.33, 70) mm, rotated rx 180 ry 0 rz 180 deg; joints [34.177, 55.495, 15.109, -144.251, 74.053, -191.188]
  Call Extruder(15390.766)
  MoveL 1573 to (-2.97, 13, 70) mm, rotated rx 180 ry 0 rz -180 deg; joints [34.384, 55.196, 15.809, -144.107, 74.419, -191.001]
  Call Extruder(15395.430)
  MoveL 1574 to (-5.78, 12.01, 70) mm, rotated rx 180 ry 0 rz -180 deg; joints [34.5, 54.874, 16.569, -144.059, 74.794, -190.766]
  Call Extruder(15400.093)
  MoveL 1575 to (-8.31, 10.42, 70) mm, rotated rx 180 ry 0 rz -180 deg; joints [34.518, 54.543, 17.35, -144.111, 75.163, -190.497]
  Call Extruder(15404.757)
  MoveL 1576 to (-10.42, 8.31, 70) mm, rotated rx 180 ry 0 rz 180 deg; joints [34.436, 54.222, 18.114, -144.263, 75.507, -190.208]
  Call Extruder(15409.421)
  MoveL 1577 to (-12.01, 5.78, 70) mm, rotated rx 180 ry 0 rz -180 deg; joints [34.254, 53.926, 18.822, -144.508, 75.81, -189.915]
  Call Extruder(15414.085)
  MoveL 1578 to (-12.99, 2.97, 70) mm, rotated rx 180 ry 0 rz -180 deg; joints [33.981, 53.669, 19.438, -144.838, 76.057, -189.634]
  Call Extruder(15418.749)
  MoveL 1579 to (-13.33, 0, 70) mm, rotated rx 180 ry 0 rz 180 deg; joints [33.63, 53.465, 19.931, -145.236, 76.235, -189.378]
  Call Extruder(15423.413)
  MoveL 1580 to (-13, -2.97, 70) mm, rotated rx -180 ry 0 rz -180 deg; joints [33.218, 53.322, 20.276, -145.683, 76.336, -189.16]
  Call Extruder(15428.076)
  MoveL 1581 to (-12.01, -5.78, 70) mm, rotated rx 180 ry 0 rz 180 deg; joints [32.767, 53.247, 20.456, -146.155, 76.352, -188.991]
  Call Extruder(15432.740)
  MoveL 1582 to (-10.42, -8.31, 70) mm, rotated rx 180 ry 0 rz 180 deg; joints [32.302, 53.245, 20.461, -146.628, 76.282, -188.878]
  Call Extruder(15437.404)
  MoveL 1583 to (-8.31, -10.42, 70) mm, rotated rx 180 ry 0 rz -180 deg; joints [31.85, 53.315, 20.292, -147.074, 76.129, -188.824]
  Call Extruder(15442.068)
  MoveL 1584 to (-5.78, -12.01, 70) mm, rotated rx -180 ry 0 rz -180 deg; joints [31.435, 53.454, 19.955, -147.47, 75.9, -188.832]
  Call Extruder(15446.731)
  MoveL 1585 to (-2.97, -12.99, 70) mm, rotated rx 180 ry 0 rz -180 deg; joints [31.079, 53.656, 19.47, -147.795, 75.605, -188.899]
  Call Extruder(15451.395)
  MoveL 1586 to (0, -13.33, 70) mm, rotated rx 180 ry 0 rz 180 deg; joints [30.801, 53.91, 18.861, -148.029, 75.26, -189.023]
  Call Extruder(15452.086)
  MoveL 1587 to (0.44, -13.28, 70) mm, rotated rx 180 ry 0 rz 180 deg; joints [30.773, 53.953, 18.757, -148.049, 75.205, -189.049]
  Set speed (130.0 mm/s)
  MoveL 1588 to (0.44, -13.28, 75) mm, rotated rx -180 ry 0 rz -180 deg; joints [30.773, 53.035, 19.122, -147.971, 74.736, -189.352]
  MoveL 1589 to (-26.25, -4.54, 75) mm, rotated rx 180 ry 0 rz 180 deg; joints [34.172, 51.147, 23.639, -144.871, 77.46, -188.685]
  Call Extruder(15454.319)
  Set speed (60.0 mm/s)
  MoveL 1590 to (-26.09, -5.96, 75) mm, rotated rx 180 ry 0 rz -180 deg; joints [33.969, 51.079, 23.803, -145.09, 77.509, -188.584]
  Call Extruder(15463.684)
  MoveL 1591 to (-24.12, -11.61, 75) mm, rotated rx -180 ry 0 rz 180 deg; joints [33.033, 50.93, 24.168, -146.065, 77.549, -188.254]
  Call Extruder(15473.049)
  MoveL 1592 to (-20.93, -16.69, 75) mm, rotated rx -180 ry 0 rz 180 deg; joints [32.066, 50.925, 24.179, -147.047, 77.417, -188.038]
  Call Extruder(15482.414)
  MoveL 1593 to (-16.69, -20.93, 75) mm, rotated rx 180 ry 0 rz -180 deg; joints [31.126, 51.066, 23.834, -147.976, 77.115, -187.94]
  Call Extruder(15491.779)
  MoveL 1594 to (-11.61, -24.11, 75) mm, rotated rx 180 ry 0 rz -180 deg; joints [30.272, 51.347, 23.153, -148.796, 76.656, -187.958]
  Call Extruder(15501.144)
  MoveL 1595 to (-5.96, -26.09, 75) mm, rotated rx 180 ry 0 rz 180 deg; joints [29.552, 51.753, 22.172, -149.458, 76.062, -188.089]
  Call Extruder(15510.509)
  MoveL 1596 to (0, -26.77, 75) mm, rotated rx 180 ry 0 rz 180 deg; joints [29.003, 52.267, 20.941, -149.926, 75.365, -188.324]
  Call Extruder(15514.207)
  MoveL 1597 to (2.35, -26.5, 75) mm, rotated rx 180 ry 0 rz 180 deg; joints [28.862, 52.501, 20.384, -150.027, 75.065, -188.454]
  Call Extruder(15519.874)
  MoveL 1598 to (5.96, -26.09, 75) mm, rotated rx -180 ry 0 rz 180 deg; joints [28.65, 52.864, 19.524, -150.178, 74.602, -188.654]
  Call Extruder(15529.239)
  MoveL 1599 to (11.61, -24.11, 75) mm, rotated rx 180 ry 0 rz 180 deg; joints [28.503, 53.516, 17.993, -150.206, 73.816, -189.067]
  Call Extruder(15538.604)
  MoveL 1600 to (16.69, -20.93, 75) mm, rotated rx 180 ry 0 rz 180 deg; joints [28.559, 54.19, 16.424, -150.015, 73.05, -189.549]
  Call Extruder(15547.969)
  MoveL 1601 to (20.93, -16.69, 75) mm, rotated rx 180 ry 0 rz -180 deg; joints [28.808, 54.853, 14.894, -149.622, 72.343, -190.082]
  Call Extruder(15557.334)
  MoveL 1602 to (24.12, -11.61, 75) mm, rotated rx -180 ry 0 rz -180 deg; joints [29.229, 55.472, 13.479, -149.055, 71.733, -190.643]
  Call Extruder(15566.699)
  MoveL 1603 to (26.09, -5.96, 75) mm, rotated rx 180 ry 0 rz -180 deg; joints [29.796, 56.013, 12.249, -148.348, 71.252, -191.207]
  Call Extruder(15576.064)
  MoveL 1604 to (26.77, 0, 75) mm, rotated rx 180 ry 0 rz -180 deg; joints [30.482, 56.449, 11.264, -147.538, 70.923, -191.745]
  Call Extruder(15585.429)
  MoveL 1605 to (26.09, 5.96, 75) mm, rotated rx -180 ry 0 rz 180 deg; joints [31.252, 56.754, 10.576, -146.668, 70.762, -192.227]
  Call Extruder(15594.794)
  MoveL 1606 to (24.11, 11.61, 75) mm, rotated rx 180 ry 0 rz -180 deg; joints [32.076, 56.914, 10.217, -145.778, 70.774, -192.625]
  Call Extruder(15604.158)
  MoveL 1607 to (20.93, 16.69, 75) mm, rotated rx 180 ry 0 rz 180 deg; joints [32.917, 56.919, 10.207, -144.908, 70.955, -192.913]
  Call Extruder(15613.524)
  MoveL 1608 to (16.69, 20.93, 75) mm, rotated rx -180 ry 0 rz 180 deg; joints [33.742, 56.768, 10.545, -144.095, 71.293, -193.073]
  Call Extruder(15622.889)
  MoveL 1609 to (11.61, 24.12, 75) mm, rotated rx -180 ry 0 rz 180 deg; joints [34.517, 56.47, 11.215, -143.373, 71.769, -193.092]
  Call Extruder(15632.253)
  MoveL 1610 to (5.96, 26.09, 75) mm, rotated rx -180 ry 0 rz 180 deg; joints [35.208, 56.042, 12.183, -142.77, 72.356, -192.97]
  Call Extruder(15641.619)
  MoveL 1611 to (0, 26.77, 75) mm, rotated rx 180 ry 0 rz 180 deg; joints [35.784, 55.506, 13.401, -142.312, 73.025, -192.71]
  Call Extruder(15650.984)
  MoveL 1612 to (-5.96, 26.09, 75) mm, rotated rx -180 ry 0 rz -180 deg; joints [36.214, 54.891, 14.807, -142.018, 73.743, -192.329]
  Call Extruder(15660.348)
  MoveL 1613 to (-11.61, 24.12, 75) mm, rotated rx 180 ry 0 rz -180 deg; joints [36.473, 54.23, 16.332, -141.906, 74.478, -191.848]
  Call Extruder(15669.713)
  MoveL 1614 to (-16.69, 20.93, 75) mm, rotated rx 180 ry 0 rz 180 deg; joints [36.542, 53.555, 17.901, -141.986, 75.196, -191.295]
  Call Extruder(15679.079)
  MoveL 1615 to (-20.93, 16.69, 75) mm, rotated rx 180 ry 0 rz -180 deg; joints [36.407, 52.902, 19.436, -142.263, 75.866, -190.702]
  Call Extruder(15688.443)
  MoveL 1616 to (-24.12, 11.61, 75) mm, rotated rx -180 ry 0 rz 180 deg; joints [36.065, 52.3, 20.862, -142.732, 76.459, -190.102]
  Call Extruder(15697.808)
  MoveL 1617 to (-26.09, 5.96, 75) mm, rotated rx 180 ry 0 rz -180 deg; joints [35.528, 51.781, 22.106, -143.379, 76.946, -189.53]
  Call Extruder(15707.173)
  MoveL 1618 to (-26.77, 0, 75) mm, rotated rx 180 ry 0 rz -180 deg; joints [34.817, 51.367, 23.104, -144.178, 77.303, -189.015]
  Call Extruder(15711.962)
  MoveL 1619 to (-26.42, -3.05, 75) mm, rotated rx 180 ry 0 rz 180 deg; joints [34.385, 51.219, 23.464, -144.643, 77.408, -188.793]
  Set speed (130.0 mm/s)
  MoveL 1620 to (-41.86, -6.29, 75) mm, rotated rx -180 ry 0 rz -180 deg; joints [35.393, 49.772, 27.03, -143.88, 79.274, -187.735]
  Call Extruder(15716.960)
  Set speed (60.0 mm/s)
  MoveL 1621 to (-41.5, -9.47, 75) mm, rotated rx -180 ry 0 rz 180 deg; joints [34.924, 49.624, 27.402, -144.378, 79.392, -187.514]
  Call Extruder(15731.856)
  MoveL 1622 to (-38.36, -18.47, 75) mm, rotated rx 180 ry 0 rz -180 deg; joints [33.373, 49.39, 27.991, -145.98, 79.488, -187.021]
  Call Extruder(15746.751)
  MoveL 1623 to (-33.29, -26.54, 75) mm, rotated rx 180 ry 0 rz -180 deg; joints [31.763, 49.383, 28.008, -147.608, 79.304, -186.716]
  Call Extruder(15761.647)
  MoveL 1624 to (-26.54, -33.28, 75) mm, rotated rx 180 ry 0 rz -180 deg; joints [30.206, 49.604, 27.452, -149.149, 78.838, -186.596]
  Call Extruder(15776.543)
  MoveL 1625 to (-18.47, -38.36, 75) mm, rotated rx 180 ry 0 rz 180 deg; joints [28.808, 50.042, 26.355, -150.499, 78.107, -186.651]
  Call Extruder(15791.439)
  MoveL 1626 to (-9.47, -41.5, 75) mm, rotated rx 180 ry 0 rz 180 deg; joints [27.654, 50.681, 24.778, -151.572, 77.15, -186.865]
  Call Extruder(15806.335)
  MoveL 1627 to (0, -42.57, 75) mm, rotated rx -180 ry 0 rz -180 deg; joints [26.805, 51.49, 22.807, -152.308, 76.021, -187.226]
  Call Extruder(15812.798)
  MoveL 1628 to (4.11, -42.11, 75) mm, rotated rx 180 ry 0 rz 180 deg; joints [26.578, 51.895, 21.832, -152.473, 75.487, -187.441]
  Call Extruder(15821.231)
  MoveL 1629 to (9.47, -41.5, 75) mm, rotated rx 180 ry 0 rz -180 deg; joints [26.29, 52.433, 20.546, -152.677, 74.785, -187.722]
  Call Extruder(15836.126)
  MoveL 1630 to (18.47, -38.36, 75) mm, rotated rx -180 ry 0 rz 180 deg; joints [26.114, 53.467, 18.107, -152.675, 73.512, -188.342]
  Call Extruder(15851.022)
  MoveL 1631 to (26.54, -33.28, 75) mm, rotated rx 180 ry 0 rz -180 deg; joints [26.262, 54.541, 15.612, -152.321, 72.274, -189.074]
  Call Extruder(15865.918)
  MoveL 1632 to (33.28, -26.54, 75) mm, rotated rx 180 ry 0 rz 180 deg; joints [26.703, 55.603, 13.181, -151.649, 71.138, -189.896]
  Call Extruder(15880.814)
  MoveL 1633 to (38.36, -18.47, 75) mm, rotated rx 180 ry 0 rz 180 deg; joints [27.4, 56.597, 10.93, -150.71, 70.162, -190.778]
  Call Extruder(15895.709)
  MoveL 1634 to (41.51, -9.47, 75) mm, rotated rx 180 ry 0 rz -180 deg; joints [28.309, 57.471, 8.971, -149.561, 69.398, -191.682]
  Call Extruder(15910.605)
  MoveL 1635 to (42.57, 0, 75) mm, rotated rx -180 ry 0 rz -180 deg; joints [29.382, 58.178, 7.4, -148.267, 68.883, -192.56]
  Call Extruder(15925.501)
  MoveL 1636 to (41.5, 9.47, 75) mm, rotated rx 180 ry 0 rz -180 deg; joints [30.575, 58.676, 6.299, -146.895, 68.641, -193.359]
  Call Extruder(15940.397)
  MoveL 1637 to (38.36, 18.47, 75) mm, rotated rx 180 ry 0 rz -180 deg; joints [31.839, 58.936, 5.724, -145.508, 68.679, -194.026]
  Call Extruder(15955.293)
  MoveL 1638 to (33.28, 26.54, 75) mm, rotated rx -180 ry 0 rz -180 deg; joints [33.128, 58.944, 5.707, -144.167, 68.99, -194.515]
  Call Extruder(15970.188)
  MoveL 1639 to (26.54, 33.29, 75) mm, rotated rx -180 ry 0 rz -180 deg; joints [34.394, 58.698, 6.25, -142.923, 69.548, -194.791]
  Call Extruder(15985.084)
  MoveL 1640 to (18.47, 38.36, 75) mm, rotated rx 180 ry 0 rz -180 deg; joints [35.592, 58.213, 7.321, -141.821, 70.319, -194.833]
  Call Extruder(15999.980)
  MoveL 1641 to (9.47, 41.51, 75) mm, rotated rx 180 ry 0 rz -180 deg; joints [36.675, 57.518, 8.867, -140.897, 71.259, -194.635]
  Call Extruder(16014.876)
  MoveL 1642 to (0, 42.57, 75) mm, rotated rx 180 ry 0 rz 180 deg; joints [37.594, 56.652, 10.806, -140.184, 72.316, -194.21]
  Call Extruder(16029.772)
  MoveL 1643 to (-9.47, 41.51, 75) mm, rotated rx -180 ry 0 rz -180 deg; joints [38.304, 55.664, 13.042, -139.71, 73.442, -193.582]
  Call Extruder(16044.667)
  MoveL 1644 to (-18.47, 38.36, 75) mm, rotated rx 180 ry 0 rz 180 deg; joints [38.762, 54.605, 15.466, -139.5, 74.587, -192.789]
  Call Extruder(16059.563)
  MoveL 1645 to (-26.54, 33.29, 75) mm, rotated rx -180 ry 0 rz -180 deg; joints [38.928, 53.53, 17.961, -139.576, 75.702, -191.879]
  Call Extruder(16074.459)
  MoveL 1646 to (-33.29, 26.54, 75) mm, rotated rx -180 ry 0 rz -180 deg; joints [38.772, 52.492, 20.406, -139.957, 76.746, -190.906]
  Call Extruder(16089.355)
  MoveL 1647 to (-38.36, 18.47, 75) mm, rotated rx 180 ry 0 rz -180 deg; joints [38.277, 51.542, 22.681, -140.648, 77.676, -189.927]
  Call Extruder(16104.251)
  MoveL 1648 to (-41.51, 9.47, 75) mm, rotated rx 180 ry 0 rz 180 deg; joints [37.447, 50.724, 24.672, -141.641, 78.453, -189.002]
  Call Extruder(16119.146)
  MoveL 1649 to (-42.57, 0, 75) mm, rotated rx -180 ry 0 rz -180 deg; joints [36.31, 50.075, 26.275, -142.903, 79.037, -188.184]
  Call Extruder(16126.701)
  MoveL 1650 to (-42.03, -4.8, 75) mm, rotated rx 180 ry 0 rz 180 deg; joints [35.612, 49.842, 26.854, -143.647, 79.218, -187.84]
  Set speed (130.0 mm/s)
  MoveL 1651 to (-54.1, -7.67, 75) mm, rotated rx 180 ry 0 rz 180 deg; joints [36.421, 48.757, 29.601, -143.008, 80.656, -186.974]
  Call Extruder(16130.773)
  Set speed (30.0 mm/s)
  MoveL 1652 to (-53.59, -12.23, 75) mm, rotated rx -180 ry 0 rz 180 deg; joints [35.732, 48.549, 30.139, -143.734, 80.838, -186.663]
  Call Extruder(16141.703)
  MoveL 1653 to (-49.52, -23.85, 75) mm, rotated rx 180 ry 0 rz -180 deg; joints [33.663, 48.251, 30.911, -145.86, 80.996, -186.058]
  Call Extruder(16152.634)
  MoveL 1654 to (-42.98, -34.27, 75) mm, rotated rx 180 ry 0 rz 180 deg; joints [31.506, 48.243, 30.933, -148.034, 80.786, -185.706]
  Call Extruder(16163.564)
  MoveL 1655 to (-34.27, -42.98, 75) mm, rotated rx 180 ry 0 rz 180 deg; joints [29.427, 48.523, 30.204, -150.093, 80.198, -185.593]
  Call Extruder(16174.494)
  MoveL 1656 to (-23.85, -49.53, 75) mm, rotated rx -180 ry 0 rz 180 deg; joints [27.581, 49.082, 28.77, -151.884, 79.251, -185.691]
  Call Extruder(16185.424)
  MoveL 1657 to (-12.23, -53.59, 75) mm, rotated rx -180 ry 0 rz -180 deg; joints [26.087, 49.898, 26.716, -153.285, 77.999, -185.974]
  Call Extruder(16196.354)
  MoveL 1658 to (0, -54.97, 75) mm, rotated rx -180 ry 0 rz 180 deg; joints [25.019, 50.935, 24.156, -154.221, 76.517, -186.425]
  Call Extruder(16201.260)
  MoveL 1659 to (5.49, -54.35, 75) mm, rotated rx -180 ry 0 rz 180 deg; joints [24.739, 51.472, 22.851, -154.426, 75.794, -186.699]
  Call Extruder(16207.285)
  MoveL 1660 to (12.23, -53.59, 75) mm, rotated rx 180 ry 0 rz -180 deg; joints [24.406, 52.147, 21.227, -154.661, 74.898, -187.033]
  Call Extruder(16218.215)
  MoveL 1661 to (23.85, -49.53, 75) mm, rotated rx -180 ry 0 rz -180 deg; joints [24.239, 53.48, 18.077, -154.61, 73.234, -187.796]
  Call Extruder(16229.145)
  MoveL 1662 to (34.27, -42.98, 75) mm, rotated rx 180 ry 0 rz 180 deg; joints [24.487, 54.87, 14.857, -154.102, 71.619, -188.705]
  Call Extruder(16240.075)
  MoveL 1663 to (42.98, -34.27, 75) mm, rotated rx 180 ry 0 rz 180 deg; joints [25.101, 56.248, 11.718, -153.189, 70.139, -189.742]
  Call Extruder(16251.005)
  MoveL 1664 to (49.52, -23.85, 75) mm, rotated rx 180 ry 0 rz 180 deg; joints [26.025, 57.544, 8.809, -151.941, 68.873, -190.875]
  Call Extruder(16261.936)
  MoveL 1665 to (53.59, -12.23, 75) mm, rotated rx -180 ry 0 rz -180 deg; joints [27.2, 58.688, 6.271, -150.435, 67.885, -192.055]
  Call Extruder(16272.866)
  MoveL 1666 to (54.97, 0, 75) mm, rotated rx -180 ry 0 rz 180 deg; joints [28.57, 59.616, 4.231, -148.757, 67.226, -193.215]
  Call Extruder(16283.796)
  MoveL 1667 to (53.59, 12.23, 75) mm, rotated rx 180 ry 0 rz 180 deg; joints [30.077, 60.273, 2.797, -146.994, 66.926, -194.283]
  Call Extruder(16294.726)
  MoveL 1668 to (49.53, 23.85, 75) mm, rotated rx 180 ry 0 rz 180 deg; joints [31.665, 60.618, 2.049, -145.228, 66.995, -195.181]
  Call Extruder(16305.656)
  MoveL 1669 to (42.98, 34.27, 75) mm, rotated rx 180 ry 0 rz 180 deg; joints [33.282, 60.628, 2.027, -143.535, 67.418, -195.843]
  Call Extruder(16316.587)
  MoveL 1670 to (34.27, 42.98, 75) mm, rotated rx -180 ry 0 rz 180 deg; joints [34.874, 60.302, 2.734, -141.977, 68.161, -196.219]
  Call Extruder(16327.517)
  MoveL 1671 to (23.85, 49.53, 75) mm, rotated rx 180 ry 0 rz 180 deg; joints [36.387, 59.663, 4.129, -140.602, 69.174, -196.278]
  Call Extruder(16338.447)
  MoveL 1672 to (12.23, 53.59, 75) mm, rotated rx 180 ry 0 rz 180 deg; joints [37.766, 58.749, 6.136, -139.449, 70.396, -196.018]
  Call Extruder(16349.377)
  MoveL 1673 to (0, 54.97, 75) mm, rotated rx 180 ry 0 rz 180 deg; joints [38.954, 57.616, 8.648, -138.55, 71.759, -195.454]
  Call Extruder(16360.307)
  MoveL 1674 to (-12.23, 53.59, 75) mm, rotated rx 180 ry 0 rz 180 deg; joints [39.895, 56.327, 11.539, -137.934, 73.198, -194.622]
  Call Extruder(16371.238)
  MoveL 1675 to (-23.85, 49.52, 75) mm, rotated rx 180 ry 0 rz 180 deg; joints [40.528, 54.952, 14.668, -137.634, 74.651, -193.572]
  Call Extruder(16382.168)
  MoveL 1676 to (-34.27, 42.98, 75) mm, rotated rx 180 ry 0 rz 180 deg; joints [40.799, 53.561, 17.888, -137.683, 76.064, -192.368]
  Call Extruder(16393.098)
  MoveL 1677 to (-42.98, 34.27, 75) mm, rotated rx 180 ry 0 rz 180 deg; joints [40.659, 52.223, 21.047, -138.113, 77.386, -191.081]
  Call Extruder(16404.028)
  MoveL 1678 to (-49.53, 23.85, 75) mm, rotated rx 180 ry 0 rz 180 deg; joints [40.072, 51.002, 23.992, -138.946, 78.572, -189.791]
  Call Extruder(16414.958)
  MoveL 1679 to (-53.59, 12.23, 75) mm, rotated rx -180 ry 0 rz 180 deg; joints [39.031, 49.953, 26.578, -140.185, 79.576, -188.577]
  Call Extruder(16425.889)
  MoveL 1680 to (-54.97, 0, 75) mm, rotated rx 180 ry 0 rz -180 deg; joints [37.56, 49.124, 28.666, -141.804, 80.348, -187.515]
  Call Extruder(16431.414)
  MoveL 1681 to (-54.27, -6.18, 75) mm, rotated rx 180 ry 0 rz -180 deg; joints [36.644, 48.827, 29.423, -142.773, 80.596, -187.077]
  Set speed (130.0 mm/s)
  MoveL 1682 to (-49.9, -9.51, 75) mm, rotated rx 180 ry 0 rz -180 deg; joints [35.741, 48.973, 29.05, -143.659, 80.303, -187.064]
  MoveL 1683 to (0.86, -13.23, 75) mm, rotated rx 180 ry 0 rz 180 deg; joints [30.747, 53.077, 19.023, -147.989, 74.684, -189.376]
  Call Extruder(16434.731)
  Set speed (80.0 mm/s)
  MoveL 1684 to (2.97, -13, 75) mm, rotated rx 180 ry 0 rz 180 deg; joints [30.614, 53.29, 18.522, -148.083, 74.418, -189.498]
  Call Extruder(16439.394)
  MoveL 1685 to (5.78, -12.01, 75) mm, rotated rx 180 ry 0 rz -180 deg; joints [30.526, 53.615, 17.761, -148.109, 74.033, -189.713]
  Call Extruder(16444.058)
  MoveL 1686 to (8.31, -10.42, 75) mm, rotated rx 180 ry 0 rz 180 deg; joints [30.538, 53.951, 16.979, -148.027, 73.656, -189.963]
  Call Extruder(16448.722)
  MoveL 1687 to (10.42, -8.31, 75) mm, rotated rx -180 ry 0 rz 180 deg; joints [30.649, 54.28, 16.217, -147.845, 73.308, -190.235]
  Call Extruder(16453.386)
  MoveL 1688 to (12.01, -5.78, 75) mm, rotated rx 180 ry 0 rz -180 deg; joints [30.85, 54.585, 15.511, -147.574, 73.006, -190.518]
  Call Extruder(16458.049)
  MoveL 1689 to (12.99, -2.97, 75) mm, rotated rx 180 ry 0 rz 180 deg; joints [31.131, 54.852, 14.898, -147.228, 72.766, -190.798]
  Call Extruder(16462.713)
  MoveL 1690 to (13.33, 0, 75) mm, rotated rx 180 ry 0 rz -180 deg; joints [31.476, 55.065, 14.408, -146.826, 72.599, -191.062]
  Call Extruder(16467.377)
  MoveL 1691 to (13, 2.97, 75) mm, rotated rx 180 ry 0 rz 180 deg; joints [31.869, 55.215, 14.065, -146.389, 72.514, -191.294]
  Call Extruder(16472.041)
  MoveL 1692 to (12.01, 5.78, 75) mm, rotated rx 180 ry 0 rz 180 deg; joints [32.292, 55.293, 13.887, -145.936, 72.514, -191.483]
  Call Extruder(16476.704)
  MoveL 1693 to (10.42, 8.31, 75) mm, rotated rx 180 ry 0 rz 180 deg; joints [32.725, 55.295, 13.881, -145.491, 72.599, -191.619]
  Call Extruder(16481.369)
  MoveL 1694 to (8.31, 10.42, 75) mm, rotated rx 180 ry 0 rz 180 deg; joints [33.149, 55.222, 14.05, -145.073, 72.762, -191.692]
  Call Extruder(16486.032)
  MoveL 1695 to (5.78, 12.01, 75) mm, rotated rx -180 ry 0 rz -180 deg; joints [33.544, 55.076, 14.384, -144.701, 72.996, -191.698]
  Call Extruder(16490.696)
  MoveL 1696 to (2.97, 12.99, 75) mm, rotated rx 180 ry 0 rz 180 deg; joints [33.893, 54.866, 14.866, -144.392, 73.288, -191.636]
  Call Extruder(16495.360)
  MoveL 1697 to (0, 13.33, 75) mm, rotated rx 180 ry 0 rz 180 deg; joints [34.177, 54.602, 15.472, -144.161, 73.624, -191.51]
  Call Extruder(16500.024)
  MoveL 1698 to (-2.97, 13, 75) mm, rotated rx 180 ry 0 rz -180 deg; joints [34.384, 54.299, 16.173, -144.018, 73.986, -191.326]
  Call Extruder(16504.687)
  MoveL 1699 to (-5.78, 12.01, 75) mm, rotated rx 180 ry 0 rz -180 deg; joints [34.5, 53.971, 16.933, -143.972, 74.358, -191.095]
  Call Extruder(16509.351)
  MoveL 1700 to (-8.31, 10.42, 75) mm, rotated rx 180 ry 0 rz -180 deg; joints [34.518, 53.635, 17.715, -144.025, 74.723, -190.827]
  Call Extruder(16514.015)
  MoveL 1701 to (-10.42, 8.31, 75) mm, rotated rx 180 ry 0 rz -180 deg; joints [34.436, 53.309, 18.479, -144.178, 75.062, -190.54]
  Call Extruder(16518.679)
  MoveL 1702 to (-12.01, 5.78, 75) mm, rotated rx 180 ry 0 rz 180 deg; joints [34.254, 53.007, 19.187, -144.426, 75.36, -190.247]
  Call Extruder(16523.342)
  MoveL 1703 to (-13, 2.97, 75) mm, rotated rx 180 ry 0 rz -180 deg; joints [33.981, 52.746, 19.803, -144.757, 75.601, -189.965]
  Call Extruder(16528.006)
  MoveL 1704 to (-13.33, 0, 75) mm, rotated rx -180 ry 0 rz -180 deg; joints [33.63, 52.538, 20.297, -145.156, 75.775, -189.707]
  Call Extruder(16532.670)
  MoveL 1705 to (-13, -2.97, 75) mm, rotated rx -180 ry 0 rz -180 deg; joints [33.218, 52.393, 20.643, -145.604, 75.871, -189.487]
  Call Extruder(16537.334)
  MoveL 1706 to (-12.01, -5.78, 75) mm, rotated rx 180 ry 0 rz -180 deg; joints [32.767, 52.317, 20.823, -146.077, 75.884, -189.315]
  Call Extruder(16541.997)
  MoveL 1707 to (-10.42, -8.31, 75) mm, rotated rx -180 ry 0 rz -180 deg; joints [32.302, 52.315, 20.828, -146.55, 75.812, -189.198]
  Call Extruder(16546.662)
  MoveL 1708 to (-8.31, -10.42, 75) mm, rotated rx 180 ry 0 rz -180 deg; joints [31.85, 52.386, 20.658, -146.997, 75.657, -189.14]
  Call Extruder(16551.325)
  MoveL 1709 to (-5.78, -12.01, 75) mm, rotated rx -180 ry 0 rz -180 deg; joints [31.435, 52.528, 20.322, -147.393, 75.427, -189.143]
  Call Extruder(16555.989)
  MoveL 1710 to (-2.97, -12.99, 75) mm, rotated rx 180 ry 0 rz 180 deg; joints [31.079, 52.732, 19.836, -147.717, 75.134, -189.207]
  Call Extruder(16560.653)
  MoveL 1711 to (0, -13.33, 75) mm, rotated rx 180 ry 0 rz -180 deg; joints [30.801, 52.991, 19.226, -147.951, 74.791, -189.327]
  Call Extruder(16562.000)
  MoveL 1712 to (0.86, -13.23, 75) mm, rotated rx 180 ry 0 rz 180 deg; joints [30.747, 53.077, 19.023, -147.989, 74.684, -189.376]
  Set speed (130.0 mm/s)
  MoveL 1713 to (0.86, -13.23, 80) mm, rotated rx 180 ry 0 rz 180 deg; joints [30.747, 52.164, 19.372, -147.906, 74.205, -189.687]
  MoveL 1714 to (-26.25, -4.54, 80) mm, rotated rx -180 ry 0 rz 180 deg; joints [34.172, 50.198, 23.991, -144.794, 76.972, -189.037]
  Call Extruder(16564.233)
  Set speed (60.0 mm/s)
  MoveL 1715 to (-26.09, -5.96, 80) mm, rotated rx -180 ry 0 rz -180 deg; joints [33.969, 50.129, 24.156, -145.012, 77.019, -188.934]
  Call Extruder(16573.598)
  MoveL 1716 to (-24.12, -11.61, 80) mm, rotated rx 180 ry 0 rz 180 deg; joints [33.033, 49.976, 24.521, -145.989, 77.052, -188.598]
  Call Extruder(16582.963)
  MoveL 1717 to (-20.93, -16.69, 80) mm, rotated rx 180 ry 0 rz 180 deg; joints [32.066, 49.972, 24.532, -146.972, 76.914, -188.373]
  Call Extruder(16592.328)
  MoveL 1718 to (-16.69, -20.93, 80) mm, rotated rx 180 ry 0 rz 180 deg; joints [31.126, 50.116, 24.187, -147.902, 76.609, -188.266]
  Call Extruder(16601.693)
  MoveL 1719 to (-11.61, -24.11, 80) mm, rotated rx 180 ry 0 rz -180 deg; joints [30.272, 50.402, 23.505, -148.721, 76.149, -188.275]
  Call Extruder(16611.057)
  MoveL 1720 to (-5.96, -26.09, 80) mm, rotated rx -180 ry 0 rz -180 deg; joints [29.552, 50.817, 22.523, -149.383, 75.558, -188.396]
  Call Extruder(16620.423)
  MoveL 1721 to (0, -26.77, 80) mm, rotated rx 180 ry 0 rz 180 deg; joints [29.003, 51.34, 21.291, -149.849, 74.866, -188.623]
  Call Extruder(16623.026)
  MoveL 1722 to (1.66, -26.58, 80) mm, rotated rx 180 ry 0 rz -180 deg; joints [28.904, 51.508, 20.898, -149.92, 74.656, -188.714]
  Call Extruder(16629.788)
  MoveL 1723 to (5.96, -26.09, 80) mm, rotated rx 180 ry 0 rz -180 deg; joints [28.65, 51.948, 19.873, -150.099, 74.11, -188.947]
  Call Extruder(16639.153)
  MoveL 1724 to (11.61, -24.12, 80) mm, rotated rx -180 ry 0 rz -180 deg; joints [28.503, 52.611, 18.341, -150.124, 73.333, -189.356]
  Call Extruder(16648.517)
  MoveL 1725 to (16.69, -20.93, 80) mm, rotated rx 180 ry 0 rz -180 deg; joints [28.559, 53.296, 16.771, -149.93, 72.575, -189.836]
  Call Extruder(16657.883)
  MoveL 1726 to (20.93, -16.69, 80) mm, rotated rx 180 ry 0 rz 180 deg; joints [28.808, 53.969, 15.24, -149.534, 71.879, -190.368]
  Call Extruder(16667.248)
  MoveL 1727 to (24.12, -11.61, 80) mm, rotated rx 180 ry 0 rz -180 deg; joints [29.229, 54.596, 13.825, -148.964, 71.279, -190.931]
  Call Extruder(16676.612)
  MoveL 1728 to (26.09, -5.96, 80) mm, rotated rx 180 ry 0 rz 180 deg; joints [29.796, 55.144, 12.595, -148.253, 70.808, -191.497]
  Call Extruder(16685.977)
  MoveL 1729 to (26.77, 0, 80) mm, rotated rx -180 ry 0 rz -180 deg; joints [30.482, 55.585, 11.611, -147.441, 70.488, -192.039]
  Call Extruder(16695.343)
  MoveL 1730 to (26.09, 5.96, 80) mm, rotated rx 180 ry 0 rz 180 deg; joints [31.252, 55.895, 10.922, -146.568, 70.334, -192.526]
  Call Extruder(16704.707)
  MoveL 1731 to (24.11, 11.61, 80) mm, rotated rx -180 ry 0 rz 180 deg; joints [32.076, 56.057, 10.564, -145.676, 70.352, -192.93]
  Call Extruder(16714.072)
  MoveL 1732 to (20.93, 16.69, 80) mm, rotated rx 180 ry 0 rz 180 deg; joints [32.917, 56.061, 10.553, -144.805, 70.537, -193.224]
  Call Extruder(16723.437)
  MoveL 1733 to (16.69, 20.93, 80) mm, rotated rx -180 ry 0 rz 180 deg; joints [33.742, 55.909, 10.892, -143.992, 70.878, -193.391]
  Call Extruder(16732.802)
  MoveL 1734 to (11.61, 24.12, 80) mm, rotated rx 180 ry 0 rz -180 deg; joints [34.517, 55.607, 11.562, -143.27, 71.355, -193.418]
  Call Extruder(16742.167)
  MoveL 1735 to (5.96, 26.09, 80) mm, rotated rx 180 ry 0 rz 180 deg; joints [35.208, 55.174, 12.53, -142.668, 71.941, -193.302]
  Call Extruder(16751.532)
  MoveL 1736 to (0, 26.77, 80) mm, rotated rx 180 ry 0 rz 180 deg; joints [35.784, 54.631, 13.747, -142.212, 72.607, -193.049]
  Call Extruder(16760.897)
  MoveL 1737 to (-5.96, 26.09, 80) mm, rotated rx 180 ry 0 rz 180 deg; joints [36.214, 54.007, 15.153, -141.92, 73.32, -192.674]
  Call Extruder(16770.262)
  MoveL 1738 to (-11.61, 24.12, 80) mm, rotated rx 180 ry 0 rz 180 deg; joints [36.473, 53.336, 16.679, -141.811, 74.048, -192.199]
  Call Extruder(16779.627)
  MoveL 1739 to (-16.69, 20.93, 80) mm, rotated rx -180 ry 0 rz -180 deg; joints [36.542, 52.651, 18.248, -141.894, 74.758, -191.65]
  Call Extruder(16788.992)
  MoveL 1740 to (-20.93, 16.69, 80) mm, rotated rx 180 ry 0 rz 180 deg; joints [36.407, 51.986, 19.785, -142.174, 75.418, -191.06]
  Call Extruder(16798.357)
  MoveL 1741 to (-24.12, 11.61, 80) mm, rotated rx -180 ry 0 rz 180 deg; joints [36.065, 51.374, 21.212, -142.647, 76, -190.462]
  Call Extruder(16807.722)
  MoveL 1742 to (-26.09, 5.96, 80) mm, rotated rx 180 ry 0 rz -180 deg; joints [35.528, 50.845, 22.456, -143.297, 76.476, -189.889]
  Call Extruder(16817.087)
  MoveL 1743 to (-26.77, 0, 80) mm, rotated rx 180 ry 0 rz 180 deg; joints [34.817, 50.423, 23.455, -144.098, 76.823, -189.371]
  Call Extruder(16821.876)
  MoveL 1744 to (-26.42, -3.05, 80) mm, rotated rx 180 ry 0 rz 180 deg; joints [34.385, 50.271, 23.817, -144.565, 76.923, -189.146]
  Set speed (130.0 mm/s)
  MoveL 1745 to (-41.86, -6.3, 80) mm, rotated rx -180 ry 0 rz 180 deg; joints [35.393, 48.793, 27.387, -143.808, 78.772, -188.108]
  Call Extruder(16826.874)
  Set speed (60.0 mm/s)
  MoveL 1746 to (-41.5, -9.47, 80) mm, rotated rx 180 ry 0 rz 180 deg; joints [34.924, 48.641, 27.76, -144.308, 78.885, -187.885]
  Call Extruder(16841.769)
  MoveL 1747 to (-38.36, -18.47, 80) mm, rotated rx 180 ry 0 rz 180 deg; joints [33.373, 48.402, 28.35, -145.913, 78.966, -187.379]
  Call Extruder(16856.665)
  MoveL 1748 to (-33.29, -26.54, 80) mm, rotated rx -180 ry 0 rz 180 deg; joints [31.763, 48.395, 28.367, -147.542, 78.773, -187.059]
  Call Extruder(16871.561)
  MoveL 1749 to (-26.54, -33.28, 80) mm, rotated rx 180 ry 0 rz -180 deg; joints [30.206, 48.621, 27.81, -149.084, 78.301, -186.923]
  Call Extruder(16886.457)
  MoveL 1750 to (-18.47, -38.36, 80) mm, rotated rx 180 ry 0 rz 180 deg; joints [28.808, 49.07, 26.711, -150.434, 77.571, -186.962]
  Call Extruder(16901.353)
  MoveL 1751 to (-9.47, -41.5, 80) mm, rotated rx 180 ry 0 rz -180 deg; joints [27.654, 49.722, 25.132, -151.505, 76.619, -187.161]
  Call Extruder(16916.248)
  MoveL 1752 to (0, -42.57, 80) mm, rotated rx 180 ry 0 rz -180 deg; joints [26.805, 50.548, 23.159, -152.239, 75.498, -187.509]
  Call Extruder(16921.617)
  MoveL 1753 to (3.41, -42.19, 80) mm, rotated rx 180 ry 0 rz 180 deg; joints [26.616, 50.891, 22.349, -152.375, 75.059, -187.684]
  Call Extruder(16931.144)
  MoveL 1754 to (9.47, -41.5, 80) mm, rotated rx -180 ry 0 rz -180 deg; joints [26.29, 51.51, 20.895, -152.604, 74.275, -187.996]
  Call Extruder(16946.040)
  MoveL 1755 to (18.47, -38.36, 80) mm, rotated rx 180 ry 0 rz -180 deg; joints [26.114, 52.561, 18.455, -152.598, 73.017, -188.61]
  Call Extruder(16960.936)
  MoveL 1756 to (26.54, -33.28, 80) mm, rotated rx 180 ry 0 rz 180 deg; joints [26.262, 53.652, 15.959, -152.239, 71.794, -189.339]
  Call Extruder(16975.832)
  MoveL 1757 to (33.28, -26.54, 80) mm, rotated rx 180 ry 0 rz 180 deg; joints [26.703, 54.729, 13.527, -151.562, 70.673, -190.161]
  Call Extruder(16990.727)
  MoveL 1758 to (38.36, -18.47, 80) mm, rotated rx -180 ry 0 rz 180 deg; joints [27.4, 55.736, 11.277, -150.618, 69.713, -191.047]
  Call Extruder(17005.623)
  MoveL 1759 to (41.5, -9.47, 80) mm, rotated rx 180 ry 0 rz -180 deg; joints [28.309, 56.62, 9.318, -149.464, 68.963, -191.956]
  Call Extruder(17020.519)
  MoveL 1760 to (42.57, 0, 80) mm, rotated rx 180 ry 0 rz -180 deg; joints [29.382, 57.334, 7.748, -148.165, 68.462, -192.84]
  Call Extruder(17035.415)
  MoveL 1761 to (41.51, 9.47, 80) mm, rotated rx 180 ry 0 rz -180 deg; joints [30.575, 57.838, 6.647, -146.789, 68.231, -193.647]
  Call Extruder(17050.311)
  MoveL 1762 to (38.36, 18.47, 80) mm, rotated rx 180 ry 0 rz 180 deg; joints [31.839, 58.101, 6.073, -145.399, 68.279, -194.323]
  Call Extruder(17065.206)
  MoveL 1763 to (33.28, 26.54, 80) mm, rotated rx 180 ry 0 rz -180 deg; joints [33.128, 58.108, 6.056, -144.056, 68.596, -194.821]
  Call Extruder(17080.102)
  MoveL 1764 to (26.54, 33.28, 80) mm, rotated rx -180 ry 0 rz -180 deg; joints [34.394, 57.86, 6.598, -142.812, 69.158, -195.107]
  Call Extruder(17094.998)
  MoveL 1765 to (18.47, 38.36, 80) mm, rotated rx 180 ry 0 rz -180 deg; joints [35.592, 57.37, 7.669, -141.71, 69.931, -195.158]
  Call Extruder(17109.894)
  MoveL 1766 to (9.47, 41.51, 80) mm, rotated rx 180 ry 0 rz -180 deg; joints [36.675, 56.667, 9.214, -140.788, 70.868, -194.971]
  Call Extruder(17124.790)
  MoveL 1767 to (0, 42.57, 80) mm, rotated rx 180 ry 0 rz -180 deg; joints [37.594, 55.792, 11.152, -140.078, 71.922, -194.556]
  Call Extruder(17139.685)
  MoveL 1768 to (-9.47, 41.5, 80) mm, rotated rx 180 ry 0 rz 180 deg; joints [38.304, 54.79, 13.388, -139.607, 73.041, -193.938]
  Call Extruder(17154.581)
  MoveL 1769 to (-18.47, 38.36, 80) mm, rotated rx -180 ry 0 rz -180 deg; joints [38.762, 53.716, 15.813, -139.401, 74.175, -193.155]
  Call Extruder(17169.477)
  MoveL 1770 to (-26.54, 33.29, 80) mm, rotated rx 180 ry 0 rz -180 deg; joints [38.928, 52.625, 18.309, -139.483, 75.278, -192.253]
  Call Extruder(17184.373)
  MoveL 1771 to (-33.29, 26.54, 80) mm, rotated rx -180 ry 0 rz -180 deg; joints [38.772, 51.569, 20.755, -139.869, 76.307, -191.286]
  Call Extruder(17199.269)
  MoveL 1772 to (-38.36, 18.47, 80) mm, rotated rx -180 ry 0 rz 180 deg; joints [38.277, 50.601, 23.033, -140.565, 77.22, -190.311]
  Call Extruder(17214.164)
  MoveL 1773 to (-41.51, 9.47, 80) mm, rotated rx -180 ry 0 rz 180 deg; joints [37.447, 49.766, 25.026, -141.563, 77.979, -189.385]
  Call Extruder(17229.060)
  MoveL 1774 to (-42.57, 0, 80) mm, rotated rx -180 ry 0 rz -180 deg; joints [36.31, 49.103, 26.631, -142.83, 78.546, -188.563]
  Call Extruder(17236.614)
  MoveL 1775 to (-42.03, -4.8, 80) mm, rotated rx 180 ry 0 rz -180 deg; joints [35.612, 48.865, 27.211, -143.575, 78.718, -188.215]
  Set speed (130.0 mm/s)
  MoveL 1776 to (-54.1, -7.67, 80) mm, rotated rx -180 ry 0 rz -180 deg; joints [36.421, 47.753, 29.963, -142.943, 80.143, -187.366]
  Call Extruder(17240.687)
  Set speed (30.0 mm/s)
  MoveL 1777 to (-53.59, -12.23, 80) mm, rotated rx 180 ry 0 rz 180 deg; joints [35.732, 47.539, 30.502, -143.67, 80.316, -187.052]
  Call Extruder(17251.617)
  MoveL 1778 to (-49.53, -23.85, 80) mm, rotated rx 180 ry 0 rz -180 deg; joints [33.663, 47.233, 31.275, -145.8, 80.455, -186.43]
  Call Extruder(17262.547)
  MoveL 1779 to (-42.98, -34.27, 80) mm, rotated rx 180 ry 0 rz -180 deg; joints [31.506, 47.225, 31.297, -147.976, 80.232, -186.057]
  Call Extruder(17273.478)
  MoveL 1780 to (-34.27, -42.98, 80) mm, rotated rx -180 ry 0 rz -180 deg; joints [29.427, 47.513, 30.567, -150.036, 79.636, -185.921]
  Call Extruder(17284.408)
  MoveL 1781 to (-23.85, -49.53, 80) mm, rotated rx -180 ry 0 rz -180 deg; joints [27.581, 48.087, 29.13, -151.825, 78.69, -185.997]
  Call Extruder(17295.338)
  MoveL 1782 to (-12.23, -53.59, 80) mm, rotated rx 180 ry 0 rz -180 deg; joints [26.087, 48.922, 27.072, -153.224, 77.446, -186.26]
  Call Extruder(17306.268)
  MoveL 1783 to (0, -54.97, 80) mm, rotated rx 180 ry 0 rz -180 deg; joints [25.019, 49.982, 24.509, -154.157, 75.977, -186.694]
  Call Extruder(17314.479)
  MoveL 1784 to (9.19, -53.93, 80) mm, rotated rx 180 ry 0 rz 180 deg; joints [24.554, 50.905, 22.314, -154.49, 74.776, -187.143]
  Call Extruder(17317.198)
  MoveL 1785 to (12.23, -53.59, 80) mm, rotated rx -180 ry 0 rz -180 deg; joints [24.406, 51.218, 21.577, -154.593, 74.374, -187.291]
  Call Extruder(17328.129)
  MoveL 1786 to (23.85, -49.52, 80) mm, rotated rx 180 ry 0 rz 180 deg; joints [24.239, 52.574, 18.425, -154.537, 72.73, -188.047]
  Call Extruder(17339.059)
  MoveL 1787 to (34.27, -42.98, 80) mm, rotated rx 180 ry 0 rz -180 deg; joints [24.487, 53.985, 15.203, -154.022, 71.135, -188.953]
  Call Extruder(17349.989)
  MoveL 1788 to (42.98, -34.27, 80) mm, rotated rx -180 ry 0 rz 180 deg; joints [25.101, 55.382, 12.064, -153.103, 69.676, -189.992]
  Call Extruder(17360.919)
  MoveL 1789 to (49.52, -23.85, 80) mm, rotated rx -180 ry 0 rz -180 deg; joints [26.025, 56.694, 9.156, -151.849, 68.429, -191.13]
  Call Extruder(17371.849)
  MoveL 1790 to (53.59, -12.23, 80) mm, rotated rx 180 ry 0 rz -180 deg; joints [27.2, 57.85, 6.619, -150.336, 67.46, -192.316]
  Call Extruder(17382.780)
  MoveL 1791 to (54.97, 0, 80) mm, rotated rx 180 ry 0 rz -180 deg; joints [28.57, 58.788, 4.581, -148.652, 66.817, -193.485]
  Call Extruder(17393.710)
  MoveL 1792 to (53.59, 12.23, 80) mm, rotated rx -180 ry 0 rz -180 deg; joints [30.077, 59.45, 3.149, -146.883, 66.531, -194.563]
  Call Extruder(17404.640)
  MoveL 1793 to (49.52, 23.85, 80) mm, rotated rx 180 ry 0 rz 180 deg; joints [31.665, 59.798, 2.401, -145.114, 66.611, -195.472]
  Call Extruder(17415.570)
  MoveL 1794 to (42.98, 34.27, 80) mm, rotated rx 180 ry 0 rz -180 deg; joints [33.282, 59.808, 2.38, -143.418, 67.042, -196.145]
  Call Extruder(17426.500)
  MoveL 1795 to (34.27, 42.98, 80) mm, rotated rx 180 ry 0 rz 180 deg; joints [34.874, 59.48, 3.086, -141.859, 67.79, -196.532]
  Call Extruder(17437.431)
  MoveL 1796 to (23.85, 49.53, 80) mm, rotated rx 180 ry 0 rz 180 deg; joints [36.387, 58.835, 4.479, -140.485, 68.805, -196.604]
  Call Extruder(17448.361)
  MoveL 1797 to (12.23, 53.59, 80) mm, rotated rx 180 ry 0 rz 180 deg; joints [37.766, 57.912, 6.484, -139.335, 70.025, -196.356]
  Call Extruder(17459.291)
  MoveL 1798 to (0, 54.97, 80) mm, rotated rx 180 ry 0 rz -180 deg; joints [38.954, 56.767, 8.995, -138.439, 71.383, -195.804]
  Call Extruder(17470.221)
  MoveL 1799 to (-12.23, 53.59, 80) mm, rotated rx 180 ry 0 rz 180 deg; joints [39.895, 55.462, 11.885, -137.828, 72.813, -194.985]
  Call Extruder(17481.151)
  MoveL 1800 to (-23.85, 49.52, 80) mm, rotated rx -180 ry 0 rz 180 deg; joints [40.528, 54.068, 15.015, -137.534, 74.255, -193.948]
  Call Extruder(17492.082)
  MoveL 1801 to (-34.27, 42.98, 80) mm, rotated rx -180 ry 0 rz 180 deg; joints [40.799, 52.656, 18.236, -137.589, 75.652, -192.755]
  Call Extruder(17503.012)
  MoveL 1802 to (-42.98, 34.27, 80) mm, rotated rx 180 ry 0 rz 180 deg; joints [40.659, 51.295, 21.397, -138.025, 76.956, -191.477]
  Call Extruder(17513.942)
  MoveL 1803 to (-49.53, 23.85, 80) mm, rotated rx -180 ry 0 rz -180 deg; joints [40.072, 50.05, 24.345, -138.865, 78.121, -190.193]
  Call Extruder(17524.872)
  MoveL 1804 to (-53.59, 12.23, 80) mm, rotated rx 180 ry 0 rz -180 deg; joints [39.031, 48.978, 26.934, -140.111, 79.101, -188.98]
  Call Extruder(17535.802)
  MoveL 1805 to (-54.97, 0, 80) mm, rotated rx 180 ry 0 rz 180 deg; joints [37.56, 48.129, 29.025, -141.736, 79.849, -187.914]
  Call Extruder(17541.328)
  MoveL 1806 to (-54.27, -6.18, 80) mm, rotated rx 180 ry 0 rz -180 deg; joints [36.644, 47.825, 29.784, -142.707, 80.086, -187.47]
  Set speed (130.0 mm/s)
  MoveL 1807 to (-49.9, -9.51, 80) mm, rotated rx 180 ry 0 rz 180 deg; joints [35.741, 47.974, 29.411, -143.592, 79.789, -187.448]
  MoveL 1808 to (0.16, -13.31, 80) mm, rotated rx 180 ry 0 rz 180 deg; joints [30.791, 52.093, 19.536, -147.875, 74.292, -189.648]
  Call Extruder(17545.740)
  Set speed (80.0 mm/s)
  MoveL 1809 to (2.97, -13, 80) mm, rotated rx -180 ry 0 rz 180 deg; joints [30.614, 52.381, 18.87, -147.999, 73.942, -189.807]
  Call Extruder(17550.403)
  MoveL 1810 to (5.78, -12.01, 80) mm, rotated rx 180 ry 0 rz -180 deg; joints [30.526, 52.712, 18.108, -148.023, 73.561, -190.02]
  Call Extruder(17555.067)
  MoveL 1811 to (8.31, -10.42, 80) mm, rotated rx -180 ry 0 rz -180 deg; joints [30.538, 53.053, 17.326, -147.94, 73.189, -190.267]
  Call Extruder(17559.731)
  MoveL 1812 to (10.42, -8.31, 80) mm, rotated rx 180 ry 0 rz 180 deg; joints [30.649, 53.387, 16.563, -147.757, 72.846, -190.539]
  Call Extruder(17564.395)
  MoveL 1813 to (12.01, -5.78, 80) mm, rotated rx 180 ry 0 rz -180 deg; joints [30.85, 53.697, 15.858, -147.484, 72.549, -190.823]
  Call Extruder(17569.058)
  MoveL 1814 to (12.99, -2.97, 80) mm, rotated rx -180 ry 0 rz -180 deg; joints [31.131, 53.967, 15.245, -147.136, 72.314, -191.104]
  Call Extruder(17573.722)
  MoveL 1815 to (13.33, 0, 80) mm, rotated rx 180 ry 0 rz 180 deg; joints [31.476, 54.184, 14.754, -146.733, 72.152, -191.369]
  Call Extruder(17578.386)
  MoveL 1816 to (12.99, 2.97, 80) mm, rotated rx -180 ry 0 rz 180 deg; joints [31.869, 54.336, 14.411, -146.294, 72.071, -191.604]
  Call Extruder(17583.050)
  MoveL 1817 to (12.01, 5.78, 80) mm, rotated rx 180 ry 0 rz 180 deg; joints [32.292, 54.415, 14.233, -145.841, 72.074, -191.797]
  Call Extruder(17587.713)
  MoveL 1818 to (10.42, 8.31, 80) mm, rotated rx 180 ry 0 rz -180 deg; joints [32.725, 54.417, 14.228, -145.395, 72.161, -191.935]
  Call Extruder(17592.377)
  MoveL 1819 to (8.31, 10.42, 80) mm, rotated rx 180 ry 0 rz -180 deg; joints [33.149, 54.342, 14.396, -144.977, 72.325, -192.012]
  Call Extruder(17597.041)
  MoveL 1820 to (5.78, 12.01, 80) mm, rotated rx 180 ry 0 rz -180 deg; joints [33.544, 54.194, 14.73, -144.605, 72.56, -192.022]
  Call Extruder(17601.705)
  MoveL 1821 to (2.97, 13, 80) mm, rotated rx 180 ry 0 rz 180 deg; joints [33.893, 53.981, 15.212, -144.297, 72.851, -191.964]
  Call Extruder(17606.369)
  MoveL 1822 to (0, 13.33, 80) mm, rotated rx 180 ry 0 rz 180 deg; joints [34.177, 53.714, 15.819, -144.066, 73.185, -191.842]
  Call Extruder(17611.033)
  MoveL 1823 to (-2.97, 12.99, 80) mm, rotated rx -180 ry 0 rz 180 deg; joints [34.384, 53.406, 16.52, -143.924, 73.545, -191.661]
  Call Extruder(17615.696)
  MoveL 1824 to (-5.78, 12.01, 80) mm, rotated rx 180 ry 0 rz -180 deg; joints [34.5, 53.073, 17.28, -143.879, 73.913, -191.432]
  Call Extruder(17620.360)
  MoveL 1825 to (-8.31, 10.42, 80) mm, rotated rx 180 ry 0 rz 180 deg; joints [34.518, 52.732, 18.062, -143.935, 74.273, -191.167]
  Call Extruder(17625.024)
  MoveL 1826 to (-10.42, 8.31, 80) mm, rotated rx 180 ry 0 rz -180 deg; joints [34.436, 52.4, 18.827, -144.089, 74.608, -190.88]
  Call Extruder(17629.688)
  MoveL 1827 to (-12.01, 5.78, 80) mm, rotated rx 180 ry 0 rz 180 deg; joints [34.254, 52.094, 19.535, -144.338, 74.9, -190.588]
  Call Extruder(17634.351)
  MoveL 1828 to (-13, 2.97, 80) mm, rotated rx 180 ry 0 rz -180 deg; joints [33.981, 51.828, 20.152, -144.671, 75.137, -190.305]
  Call Extruder(17639.015)
  MoveL 1829 to (-13.33, 0, 80) mm, rotated rx 180 ry 0 rz -180 deg; joints [33.63, 51.616, 20.646, -145.072, 75.305, -190.046]
  Call Extruder(17643.679)
  MoveL 1830 to (-13, -2.97, 80) mm, rotated rx 180 ry 0 rz -180 deg; joints [33.218, 51.468, 20.992, -145.521, 75.397, -189.823]
  Call Extruder(17648.343)
  MoveL 1831 to (-12.01, -5.78, 80) mm, rotated rx -180 ry 0 rz 180 deg; joints [32.767, 51.391, 21.172, -145.995, 75.406, -189.647]
  Call Extruder(17653.006)
  MoveL 1832 to (-10.42, -8.31, 80) mm, rotated rx 180 ry 0 rz 180 deg; joints [32.302, 51.389, 21.178, -146.469, 75.331, -189.526]
  Call Extruder(17657.670)
  MoveL 1833 to (-8.31, -10.42, 80) mm, rotated rx 180 ry 0 rz -180 deg; joints [31.85, 51.461, 21.008, -146.916, 75.175, -189.464]
  Call Extruder(17662.334)
  MoveL 1834 to (-5.78, -12.01, 80) mm, rotated rx -180 ry 0 rz -180 deg; joints [31.435, 51.606, 20.671, -147.312, 74.945, -189.463]
  Call Extruder(17666.998)
  MoveL 1835 to (-2.97, -12.99, 80) mm, rotated rx 180 ry 0 rz 180 deg; joints [31.079, 51.814, 20.185, -147.635, 74.652, -189.522]
  Call Extruder(17671.662)
  MoveL 1836 to (0, -13.33, 80) mm, rotated rx 180 ry 0 rz 180 deg; joints [30.801, 52.077, 19.574, -147.868, 74.312, -189.639]
  Call Extruder(17671.914)
  MoveL 1837 to (0.16, -13.31, 80) mm, rotated rx 180 ry 0 rz 180 deg; joints [30.791, 52.093, 19.536, -147.875, 74.292, -189.648]
  Set speed (130.0 mm/s)
  MoveL 1838 to (0.16, -13.31, 85) mm, rotated rx 180 ry 0 rz -180 deg; joints [30.791, 51.184, 19.868, -147.787, 73.803, -189.968]
  MoveL 1839 to (-26.25, -4.54, 85) mm, rotated rx 180 ry 0 rz -180 deg; joints [34.172, 49.254, 24.326, -144.711, 76.475, -189.398]
  Call Extruder(17674.147)
  Set speed (60.0 mm/s)
  MoveL 1840 to (-26.09, -5.96, 85) mm, rotated rx 180 ry 0 rz -180 deg; joints [33.969, 49.184, 24.492, -144.93, 76.52, -189.294]
  Call Extruder(17683.511)
  MoveL 1841 to (-24.12, -11.61, 85) mm, rotated rx 180 ry 0 rz 180 deg; joints [33.033, 49.028, 24.857, -145.909, 76.544, -188.95]
  Call Extruder(17692.876)
  MoveL 1842 to (-20.93, -16.69, 85) mm, rotated rx 180 ry 0 rz 180 deg; joints [32.066, 49.023, 24.868, -146.893, 76.401, -188.717]
  Call Extruder(17702.242)
  MoveL 1843 to (-16.69, -20.93, 85) mm, rotated rx 180 ry 0 rz -180 deg; joints [31.126, 49.17, 24.523, -147.823, 76.092, -188.6]
  Call Extruder(17711.606)
  MoveL 1844 to (-11.61, -24.11, 85) mm, rotated rx 180 ry 0 rz -180 deg; joints [30.272, 49.462, 23.84, -148.642, 75.632, -188.599]
  Call Extruder(17720.971)
  MoveL 1845 to (-5.96, -26.09, 85) mm, rotated rx 180 ry 0 rz 180 deg; joints [29.552, 49.885, 22.856, -149.302, 75.043, -188.712]
  Call Extruder(17730.336)
  MoveL 1846 to (0, -26.77, 85) mm, rotated rx 180 ry 0 rz -180 deg; joints [29.003, 50.418, 21.623, -149.768, 74.356, -188.931]
  Call Extruder(17735.347)
  MoveL 1847 to (3.19, -26.41, 85) mm, rotated rx -180 ry 0 rz 180 deg; joints [28.813, 50.748, 20.867, -149.902, 73.957, -189.101]
  Call Extruder(17739.701)
  MoveL 1848 to (5.96, -26.09, 85) mm, rotated rx 180 ry 0 rz 180 deg; joints [28.65, 51.037, 20.204, -150.015, 73.608, -189.249]
  Call Extruder(17749.066)
  MoveL 1849 to (11.61, -24.11, 85) mm, rotated rx 180 ry 0 rz 180 deg; joints [28.503, 51.711, 18.671, -150.037, 72.839, -189.653]
  Call Extruder(17758.431)
  MoveL 1850 to (16.69, -20.93, 85) mm, rotated rx 180 ry 0 rz 180 deg; joints [28.559, 52.407, 17.1, -149.84, 72.092, -190.13]
  Call Extruder(17767.796)
  MoveL 1851 to (20.93, -16.69, 85) mm, rotated rx 180 ry 0 rz 180 deg; joints [28.808, 53.09, 15.57, -149.442, 71.405, -190.662]
  Call Extruder(17777.161)
  MoveL 1852 to (24.12, -11.61, 85) mm, rotated rx -180 ry 0 rz -180 deg; joints [29.229, 53.726, 14.154, -148.868, 70.816, -191.226]
  Call Extruder(17786.526)
  MoveL 1853 to (26.09, -5.96, 85) mm, rotated rx 180 ry 0 rz 180 deg; joints [29.796, 54.281, 12.924, -148.154, 70.354, -191.796]
  Call Extruder(17795.891)
  MoveL 1854 to (26.77, 0, 85) mm, rotated rx 180 ry 0 rz 180 deg; joints [30.482, 54.728, 11.94, -147.339, 70.043, -192.342]
  Call Extruder(17805.256)
  MoveL 1855 to (26.09, 5.96, 85) mm, rotated rx 180 ry 0 rz -180 deg; joints [31.252, 55.042, 11.252, -146.463, 69.897, -192.834]
  Call Extruder(17814.621)
  MoveL 1856 to (24.11, 11.61, 85) mm, rotated rx 180 ry 0 rz 180 deg; joints [32.076, 55.205, 10.893, -145.57, 69.921, -193.243]
  Call Extruder(17823.986)
  MoveL 1857 to (20.93, 16.69, 85) mm, rotated rx 180 ry 0 rz 180 deg; joints [32.917, 55.21, 10.883, -144.697, 70.111, -193.544]
  Call Extruder(17833.351)
  MoveL 1858 to (16.69, 20.93, 85) mm, rotated rx 180 ry 0 rz -180 deg; joints [33.742, 55.056, 11.221, -143.884, 70.455, -193.718]
  Call Extruder(17842.716)
  MoveL 1859 to (11.61, 24.12, 85) mm, rotated rx 180 ry 0 rz 180 deg; joints [34.517, 54.75, 11.891, -143.162, 70.932, -193.752]
  Call Extruder(17852.081)
  MoveL 1860 to (5.96, 26.09, 85) mm, rotated rx 180 ry 0 rz -180 deg; joints [35.208, 54.311, 12.859, -142.562, 71.517, -193.643]
  Call Extruder(17861.446)
  MoveL 1861 to (0, 26.77, 85) mm, rotated rx 180 ry 0 rz -180 deg; joints [35.784, 53.761, 14.076, -142.106, 72.18, -193.397]
  Call Extruder(17870.811)
  MoveL 1862 to (-5.96, 26.09, 85) mm, rotated rx 180 ry 0 rz -180 deg; joints [36.214, 53.129, 15.483, -141.817, 72.888, -193.029]
  Call Extruder(17880.176)
  MoveL 1863 to (-11.61, 24.12, 85) mm, rotated rx 180 ry 0 rz 180 deg; joints [36.473, 52.447, 17.008, -141.711, 73.609, -192.559]
  Call Extruder(17889.541)
  MoveL 1864 to (-16.69, 20.93, 85) mm, rotated rx -180 ry 0 rz -180 deg; joints [36.542, 51.751, 18.579, -141.797, 74.31, -192.015]
  Call Extruder(17898.906)
  MoveL 1865 to (-20.93, 16.69, 85) mm, rotated rx -180 ry 0 rz 180 deg; joints [36.407, 51.075, 20.117, -142.08, 74.961, -191.428]
  Call Extruder(17908.271)
  MoveL 1866 to (-24.12, 11.61, 85) mm, rotated rx 180 ry 0 rz 180 deg; joints [36.065, 50.453, 21.544, -142.556, 75.532, -190.831]
  Call Extruder(17917.636)
  MoveL 1867 to (-26.09, 5.96, 85) mm, rotated rx 180 ry 0 rz -180 deg; joints [35.528, 49.913, 22.79, -143.209, 75.997, -190.257]
  Call Extruder(17927.001)
  MoveL 1868 to (-26.77, 0, 85) mm, rotated rx 180 ry 0 rz 180 deg; joints [34.817, 49.484, 23.79, -144.014, 76.333, -189.736]
  Call Extruder(17931.790)
  MoveL 1869 to (-26.42, -3.05, 85) mm, rotated rx -180 ry 0 rz -180 deg; joints [34.385, 49.329, 24.152, -144.481, 76.429, -189.509]
  Set speed (130.0 mm/s)
  MoveL 1870 to (-41.86, -6.29, 85) mm, rotated rx 180 ry 0 rz -180 deg; joints [35.393, 47.818, 27.727, -143.732, 78.259, -188.491]
  Call Extruder(17936.787)
  Set speed (60.0 mm/s)
  MoveL 1871 to (-41.5, -9.47, 85) mm, rotated rx 180 ry 0 rz 180 deg; joints [34.924, 47.663, 28.1, -144.233, 78.367, -188.265]
  Call Extruder(17951.683)
  MoveL 1872 to (-38.36, -18.47, 85) mm, rotated rx 180 ry 0 rz -180 deg; joints [33.373, 47.418, 28.691, -145.841, 78.434, -187.747]
  Call Extruder(17966.579)
  MoveL 1873 to (-33.29, -26.54, 85) mm, rotated rx -180 ry 0 rz -180 deg; joints [31.763, 47.41, 28.708, -147.472, 78.23, -187.412]
  Call Extruder(17981.475)
  MoveL 1874 to (-26.54, -33.28, 85) mm, rotated rx -180 ry 0 rz -180 deg; joints [30.206, 47.642, 28.151, -149.014, 77.754, -187.259]
  Call Extruder(17996.371)
  MoveL 1875 to (-18.47, -38.36, 85) mm, rotated rx 180 ry 0 rz 180 deg; joints [28.808, 48.101, 27.05, -150.363, 77.023, -187.28]
  Call Extruder(18011.266)
  MoveL 1876 to (-9.47, -41.51, 85) mm, rotated rx 180 ry 0 rz 180 deg; joints [27.654, 48.768, 25.469, -151.433, 76.076, -187.464]
  Call Extruder(18026.162)
  MoveL 1877 to (0, -42.57, 85) mm, rotated rx 180 ry 0 rz 180 deg; joints [26.805, 49.611, 23.493, -152.165, 74.965, -187.799]
  Call Extruder(18033.938)
  MoveL 1878 to (4.95, -42.02, 85) mm, rotated rx 180 ry 0 rz -180 deg; joints [26.533, 50.118, 22.317, -152.358, 74.335, -188.049]
  Call Extruder(18041.058)
  MoveL 1879 to (9.47, -41.5, 85) mm, rotated rx 180 ry 0 rz -180 deg; joints [26.29, 50.59, 21.227, -152.527, 73.754, -188.277]
  Call Extruder(18055.954)
  MoveL 1880 to (18.47, -38.36, 85) mm, rotated rx 180 ry 0 rz 180 deg; joints [26.114, 51.66, 18.786, -152.517, 72.511, -188.885]
  Call Extruder(18070.850)
  MoveL 1881 to (26.54, -33.28, 85) mm, rotated rx 180 ry 0 rz 180 deg; joints [26.262, 52.768, 16.289, -152.152, 71.304, -189.612]
  Call Extruder(18085.745)
  MoveL 1882 to (33.28, -26.54, 85) mm, rotated rx 180 ry 0 rz 180 deg; joints [26.703, 53.86, 13.856, -151.471, 70.199, -190.434]
  Call Extruder(18100.641)
  MoveL 1883 to (38.36, -18.47, 85) mm, rotated rx 180 ry 0 rz 180 deg; joints [27.4, 54.88, 11.606, -150.521, 69.255, -191.323]
  Call Extruder(18115.537)
  MoveL 1884 to (41.51, -9.47, 85) mm, rotated rx 180 ry 0 rz 180 deg; joints [28.309, 55.775, 9.647, -149.362, 68.52, -192.237]
  Call Extruder(18130.433)
  MoveL 1885 to (42.57, 0, 85) mm, rotated rx 180 ry 0 rz 180 deg; joints [29.382, 56.497, 8.078, -148.059, 68.032, -193.128]
  Call Extruder(18145.329)
  MoveL 1886 to (41.51, 9.47, 85) mm, rotated rx 180 ry 0 rz 180 deg; joints [30.575, 57.006, 6.978, -146.678, 67.813, -193.943]
  Call Extruder(18160.224)
  MoveL 1887 to (38.36, 18.47, 85) mm, rotated rx 180 ry 0 rz -180 deg; joints [31.839, 57.272, 6.404, -145.285, 67.869, -194.628]
  Call Extruder(18175.120)
  MoveL 1888 to (33.28, 26.54, 85) mm, rotated rx 180 ry 0 rz -180 deg; joints [33.128, 57.28, 6.388, -143.94, 68.193, -195.136]
  Call Extruder(18190.016)
  MoveL 1889 to (26.54, 33.28, 85) mm, rotated rx -180 ry 0 rz 180 deg; joints [34.394, 57.029, 6.929, -142.695, 68.76, -195.431]
  Call Extruder(18204.912)
  MoveL 1890 to (18.47, 38.36, 85) mm, rotated rx 180 ry 0 rz -180 deg; joints [35.592, 56.534, 8, -141.594, 69.534, -195.493]
  Call Extruder(18219.807)
  MoveL 1891 to (9.47, 41.51, 85) mm, rotated rx -180 ry 0 rz -180 deg; joints [36.675, 55.823, 9.544, -140.674, 70.47, -195.316]
  Call Extruder(18234.703)
  MoveL 1892 to (0, 42.57, 85) mm, rotated rx 180 ry 0 rz 180 deg; joints [37.594, 54.937, 11.482, -139.967, 71.519, -194.912]
  Call Extruder(18249.599)
  MoveL 1893 to (-9.47, 41.5, 85) mm, rotated rx 180 ry 0 rz -180 deg; joints [38.304, 53.923, 13.718, -139.5, 72.631, -194.304]
  Call Extruder(18264.495)
  MoveL 1894 to (-18.47, 38.36, 85) mm, rotated rx 180 ry 0 rz 180 deg; joints [38.762, 52.833, 16.142, -139.298, 73.755, -193.53]
  Call Extruder(18279.391)
  MoveL 1895 to (-26.54, 33.29, 85) mm, rotated rx 180 ry 0 rz 180 deg; joints [38.928, 51.725, 18.639, -139.384, 74.846, -192.636]
  Call Extruder(18294.287)
  MoveL 1896 to (-33.29, 26.54, 85) mm, rotated rx 180 ry 0 rz 180 deg; joints [38.772, 50.651, 21.087, -139.775, 75.86, -191.675]
  Call Extruder(18309.182)
  MoveL 1897 to (-38.36, 18.47, 85) mm, rotated rx 180 ry 0 rz 180 deg; joints [38.277, 49.665, 23.367, -140.477, 76.756, -190.703]
  Call Extruder(18324.078)
  MoveL 1898 to (-41.51, 9.47, 85) mm, rotated rx -180 ry 0 rz -180 deg; joints [37.447, 48.813, 25.362, -141.479, 77.497, -189.778]
  Call Extruder(18338.974)
  MoveL 1899 to (-42.57, 0, 85) mm, rotated rx 180 ry 0 rz 180 deg; joints [36.31, 48.135, 26.969, -142.751, 78.045, -188.951]
  Call Extruder(18346.528)
